C09076=1067.956,264.109,-90.042,173.798,30.770,155.599
C09077=1067.962,264.356,-90.071,173.801,30.774,155.599
C09078=1067.968,264.604,-90.100,173.804,30.779,155.600
C09079=1067.974,264.852,-90.129,173.805,30.782,155.601
C09080=1067.980,265.101,-90.157,173.808,30.786,155.601
C09081=1067.986,265.349,-90.187,173.811,30.791,155.602
C09082=1067.992,265.598,-90.216,173.813,30.794,155.603
C09083=1067.998,265.846,-90.245,173.816,30.798,155.604
C09084=1068.005,266.094,-90.274,173.819,30.803,155.604
C09085=1068.010,266.342,-90.304,173.821,30.806,155.605
C09086=1068.016,266.591,-90.332,173.823,30.811,155.606
C09087=1068.022,266.838,-90.361,173.826,30.815,155.606
C09088=1068.028,267.087,-90.390,173.829,30.818,155.607
C09089=1068.033,267.335,-90.419,173.831,30.823,155.608
C09090=1068.040,267.583,-90.449,173.834,30.827,155.609
C09091=1068.046,267.831,-90.478,173.837,30.831,155.609
C09092=1068.052,268.079,-90.507,173.838,30.835,155.610
C09093=1068.058,268.328,-90.536,173.841,30.839,155.611
C09094=1068.064,268.576,-90.565,173.844,30.842,155.611
C09095=1068.070,268.824,-90.594,173.847,30.846,155.612
C09096=1068.076,269.072,-90.623,173.849,30.851,155.613
C09097=1068.082,269.321,-90.653,173.852,30.854,155.613
C09098=1068.088,269.569,-90.682,173.855,30.859,155.614
C09099=1068.094,269.817,-90.712,173.857,30.863,155.615
C09100=1068.100,270.065,-90.741,173.860,30.867,155.616
C09101=1068.106,270.314,-90.770,173.862,30.871,155.616
C09102=1068.112,270.562,-90.799,173.864,30.875,155.617
C09103=1068.118,270.810,-90.829,173.867,30.878,155.618
C09104=1068.124,271.058,-90.859,173.870,30.883,155.618
C09105=1068.130,271.306,-90.888,173.873,30.887,155.619
C09106=1068.136,271.554,-90.917,173.875,30.891,155.620
C09107=1068.142,271.803,-90.946,173.878,30.895,155.621
C09108=1068.148,272.051,-90.976,173.881,30.899,155.621
C09109=1068.154,272.299,-91.006,173.883,30.903,155.622
C09110=1068.161,272.547,-91.035,173.886,30.907,155.623
C09111=1068.166,272.796,-91.065,173.888,30.911,155.623
C09112=1068.173,273.044,-91.094,173.891,30.915,155.624
C09113=1068.178,273.292,-91.124,173.893,30.919,155.625
C09114=1068.185,273.540,-91.153,173.896,30.923,155.626
C09115=1068.190,273.788,-91.183,173.899,30.927,155.626
C09116=1068.197,274.036,-91.213,173.901,30.931,155.627
C09117=1068.202,274.284,-91.242,173.904,30.935,155.628
C09118=1068.208,274.532,-91.271,173.907,30.939,155.628
C09119=1068.214,274.780,-91.302,173.910,30.943,155.629
C09120=1068.220,275.028,-91.331,173.912,30.947,155.630
C09121=1068.227,275.278,-91.361,173.915,30.951,155.631
C09122=1068.232,275.525,-91.391,173.918,30.955,155.631
C09123=1068.239,275.774,-91.420,173.920,30.960,155.632
C09124=1068.244,275.987,-91.446,173.922,30.963,155.633
C09125=1068.249,276.202,-91.471,173.925,30.967,155.633
C09126=1068.255,276.416,-91.497,173.927,30.970,155.634
C09127=1068.259,276.630,-91.524,173.929,30.974,155.634
C09128=1068.264,276.845,-91.549,173.931,30.977,155.635
C09129=1068.270,277.059,-91.575,173.934,30.980,155.636
C09130=1068.275,277.273,-91.600,173.936,30.984,155.636
C09131=1068.280,277.487,-91.626,173.938,30.987,155.637
C09132=1068.286,277.735,-91.657,173.941,30.992,155.638
C09133=1068.292,277.983,-91.686,173.944,30.996,155.638
C09134=1068.298,278.231,-91.716,173.947,31.000,155.639
C09135=1068.304,278.480,-91.746,173.949,31.004,155.640
C09136=1068.311,278.727,-91.776,173.952,31.008,155.640
C09137=1068.316,278.976,-91.805,173.955,31.012,155.641
C09138=1068.322,279.224,-91.836,173.957,31.016,155.642
C09139=1068.328,279.472,-91.866,173.960,31.020,155.643
C09140=1068.335,279.720,-91.896,173.963,31.024,155.643
C09141=1068.340,279.968,-91.926,173.966,31.028,155.644
C09142=1068.346,280.216,-91.956,173.968,31.032,155.645
C09143=1068.353,280.464,-91.985,173.971,31.036,155.646
C09144=1068.358,280.712,-92.016,173.974,31.040,155.646
C09145=1068.365,280.961,-92.046,173.977,31.045,155.647
C09146=1068.371,281.208,-92.077,173.978,31.048,155.648
C09147=1068.376,281.457,-92.106,173.981,31.053,155.648
C09148=1068.382,281.705,-92.137,173.984,31.056,155.649
C09149=1068.388,281.953,-92.167,173.986,31.061,155.650
C09150=1068.394,282.201,-92.198,173.989,31.065,155.651
C09151=1068.400,282.449,-92.228,173.992,31.069,155.651
C09152=1068.406,282.697,-92.257,173.995,31.073,155.652
C09153=1068.412,282.945,-92.288,173.997,31.077,155.653
C09154=1068.418,283.193,-92.318,174.000,31.081,155.654
C09155=1068.424,283.441,-92.349,174.003,31.085,155.654
C09156=1068.430,283.689,-92.379,174.006,31.090,155.655
C09157=1068.436,283.937,-92.410,174.008,31.093,155.656
C09158=1068.442,284.185,-92.440,174.011,31.098,155.656
C09159=1068.448,284.433,-92.470,174.015,31.102,155.657
C09160=1068.455,284.682,-92.501,174.017,31.106,155.658
C09161=1068.460,284.929,-92.531,174.020,31.110,155.659
C09162=1068.466,285.177,-92.562,174.023,31.114,155.659
C09163=1068.473,285.426,-92.592,174.026,31.119,155.660
C09164=1068.478,285.674,-92.623,174.028,31.122,155.661
C09165=1068.484,285.921,-92.653,174.031,31.127,155.662
C09166=1068.491,286.170,-92.684,174.034,31.131,155.662
C09167=1068.496,286.418,-92.714,174.037,31.135,155.663
C09168=1068.502,286.666,-92.745,174.039,31.139,155.664
C09169=1068.509,286.914,-92.775,174.042,31.143,155.664
C09170=1068.515,287.162,-92.805,174.045,31.147,155.665
C09171=1068.521,287.409,-92.835,174.048,31.151,155.666
C09172=1068.527,287.658,-92.866,174.050,31.155,155.667
C09173=1068.533,287.906,-92.896,174.053,31.159,155.667
C09174=1068.540,288.154,-92.928,174.056,31.164,155.668
C09175=1068.546,288.401,-92.958,174.059,31.168,155.669
C09176=1068.552,288.650,-92.989,174.061,31.172,155.670
C09177=1068.558,288.898,-93.019,174.064,31.176,155.670
C09178=1068.563,289.146,-93.050,174.067,31.180,155.671
C09179=1068.570,289.394,-93.082,174.069,31.184,155.672
C09180=1068.575,289.613,-93.108,174.072,31.188,155.673
C09181=1068.580,289.832,-93.136,174.075,31.192,155.673
C09182=1068.586,290.052,-93.163,174.078,31.195,155.674
C09183=1068.591,290.271,-93.191,174.080,31.199,155.675
C09184=1068.597,290.490,-93.217,174.082,31.203,155.675
C09185=1068.602,290.710,-93.245,174.085,31.206,155.676
C09186=1068.607,290.929,-93.272,174.088,31.210,155.676
C09187=1068.613,291.149,-93.300,174.090,31.214,155.677
C09188=1068.619,291.397,-93.330,174.092,31.218,155.678
C09189=1068.625,291.645,-93.361,174.095,31.222,155.679
C09190=1068.631,291.893,-93.393,174.099,31.226,155.679
C09191=1068.636,292.141,-93.423,174.102,31.230,155.680
C09192=1068.643,292.389,-93.454,174.104,31.235,155.681
C09193=1068.649,292.636,-93.485,174.107,31.239,155.682
C09194=1068.655,292.885,-93.517,174.110,31.243,155.682
C09195=1068.661,293.132,-93.547,174.113,31.247,155.683
C09196=1068.667,293.381,-93.578,174.115,31.252,155.684
C09197=1068.673,293.628,-93.609,174.118,31.255,155.685
C09198=1068.679,293.877,-93.640,174.121,31.260,155.685
C09199=1068.685,294.124,-93.671,174.124,31.264,155.686
C09200=1068.692,294.372,-93.703,174.127,31.268,155.687
C09201=1068.697,294.620,-93.734,174.130,31.272,155.688
C09202=1068.704,294.868,-93.765,174.133,31.277,155.688
C09203=1068.710,295.117,-93.796,174.136,31.281,155.689
C09204=1068.715,295.364,-93.827,174.138,31.285,155.690
C09205=1068.722,295.612,-93.859,174.141,31.289,155.691
C09206=1068.728,295.860,-93.889,174.144,31.293,155.692
C09207=1068.734,296.108,-93.921,174.147,31.298,155.692
C09208=1068.740,296.355,-93.952,174.150,31.302,155.693
C09209=1068.746,296.604,-93.984,174.153,31.306,155.694
C09210=1068.753,296.852,-94.015,174.156,31.310,155.695
C09211=1068.759,297.099,-94.046,174.159,31.315,155.695
C09212=1068.764,297.348,-94.077,174.161,31.319,155.696
C09213=1068.770,297.595,-94.108,174.164,31.323,155.697
C09214=1068.776,297.843,-94.140,174.167,31.327,155.698
C09215=1068.782,298.091,-94.172,174.171,31.332,155.698
C09216=1068.789,298.339,-94.204,174.173,31.336,155.699
C09217=1068.794,298.586,-94.235,174.176,31.341,155.700
C09218=1068.800,298.835,-94.267,174.179,31.345,155.701
C09219=1068.806,299.083,-94.298,174.182,31.349,155.702
C09220=1068.812,299.331,-94.330,174.184,31.354,155.702
C09221=1068.818,299.579,-94.362,174.188,31.357,155.703
C09222=1068.824,299.826,-94.393,174.191,31.362,155.704
C09223=1068.830,300.074,-94.425,174.194,31.366,155.705
C09224=1068.836,300.322,-94.457,174.196,31.370,155.705
C09225=1068.842,300.570,-94.488,174.199,31.375,155.706
C09226=1068.848,300.818,-94.520,174.202,31.379,155.707
C09227=1068.853,301.065,-94.552,174.206,31.383,155.708
C09228=1068.859,301.314,-94.584,174.208,31.388,155.709
C09229=1068.866,301.562,-94.615,174.211,31.392,155.709
C09230=1068.871,301.809,-94.647,174.214,31.396,155.710
C09231=1068.877,302.057,-94.679,174.217,31.401,155.711
C09232=1068.884,302.305,-94.710,174.220,31.405,155.712
C09233=1068.890,302.553,-94.742,174.223,31.409,155.713
C09234=1068.896,302.801,-94.774,174.226,31.414,155.713
C09235=1068.902,303.049,-94.806,174.229,31.418,155.714
C09236=1068.908,303.275,-94.835,174.232,31.422,155.715
C09237=1068.913,303.502,-94.864,174.234,31.426,155.716
C09238=1068.918,303.729,-94.893,174.237,31.430,155.716
C09239=1068.924,303.956,-94.922,174.240,31.434,155.717
C09240=1068.930,304.182,-94.952,174.243,31.438,155.718
C09241=1068.935,304.409,-94.981,174.245,31.442,155.719
C09242=1068.940,304.636,-95.010,174.248,31.446,155.719
C09243=1068.946,304.863,-95.040,174.251,31.450,155.720
C09244=1068.952,305.110,-95.071,174.254,31.455,155.721
C09245=1068.958,305.359,-95.103,174.257,31.459,155.722
C09246=1068.964,305.607,-95.135,174.259,31.463,155.722
C09247=1068.971,305.854,-95.168,174.263,31.468,155.723
C09248=1068.976,306.102,-95.200,174.266,31.472,155.724
C09249=1068.983,306.350,-95.231,174.269,31.476,155.725
C09250=1068.989,306.597,-95.264,174.271,31.480,155.726
C09251=1068.995,306.846,-95.296,174.275,31.485,155.726
C09252=1069.001,307.094,-95.328,174.278,31.489,155.727
C09253=1069.007,307.341,-95.361,174.281,31.494,155.728
C09254=1069.014,307.589,-95.392,174.284,31.498,155.729
C09255=1069.020,307.836,-95.424,174.287,31.502,155.730
C09256=1069.026,308.085,-95.456,174.290,31.507,155.730
C09257=1069.032,308.332,-95.489,174.293,31.511,155.731
C09258=1069.038,308.580,-95.521,174.297,31.516,155.732
C09259=1069.045,308.828,-95.553,174.299,31.520,155.733
C09260=1069.051,309.076,-95.585,174.302,31.524,155.734
C09261=1069.057,309.324,-95.617,174.305,31.529,155.734
C09262=1069.063,309.572,-95.650,174.309,31.533,155.735
C09263=1069.069,309.819,-95.682,174.312,31.537,155.736
C09264=1069.075,310.067,-95.715,174.314,31.542,155.737
C09265=1069.081,310.314,-95.747,174.318,31.546,155.738
C09266=1069.088,310.562,-95.779,174.321,31.550,155.738
C09267=1069.094,310.810,-95.811,174.324,31.555,155.739
C09268=1069.100,311.058,-95.843,174.326,31.559,155.740
C09269=1069.107,311.306,-95.876,174.330,31.564,155.741
C09270=1069.113,311.553,-95.909,174.333,31.568,155.742
C09271=1069.119,311.801,-95.941,174.336,31.572,155.742
C09272=1069.125,312.049,-95.974,174.340,31.577,155.743
C09273=1069.132,312.297,-96.006,174.342,31.581,155.744
C09274=1069.138,312.544,-96.038,174.345,31.585,155.745
C09275=1069.145,312.792,-96.071,174.349,31.590,155.746
C09276=1069.151,313.040,-96.104,174.352,31.595,155.747
C09277=1069.158,313.288,-96.137,174.355,31.599,155.747
C09278=1069.164,313.536,-96.169,174.358,31.603,155.748
C09279=1069.170,313.784,-96.201,174.361,31.608,155.749
C09280=1069.176,314.031,-96.234,174.364,31.612,155.750
C09281=1069.183,314.279,-96.267,174.368,31.617,155.751
C09282=1069.189,314.527,-96.300,174.370,31.621,155.751
C09283=1069.194,314.775,-96.332,174.373,31.626,155.752
C09284=1069.200,315.023,-96.365,174.377,31.630,155.753
C09285=1069.207,315.270,-96.398,174.380,31.635,155.754
C09286=1069.212,315.518,-96.431,174.383,31.640,155.755
C09287=1069.219,315.766,-96.464,174.386,31.644,155.756
C09288=1069.224,316.014,-96.497,174.389,31.649,155.757
C09289=1069.230,316.261,-96.530,174.392,31.654,155.758
C09290=1069.237,316.509,-96.563,174.396,31.658,155.758
C09291=1069.242,316.757,-96.596,174.399,31.663,155.759
C09292=1069.248,316.985,-96.626,174.401,31.666,155.760
C09293=1069.253,317.214,-96.656,174.404,31.671,155.761
C09294=1069.260,317.443,-96.687,174.407,31.675,155.762
C09295=1069.265,317.671,-96.718,174.410,31.679,155.762
C09296=1069.270,317.899,-96.749,174.413,31.684,155.763
C09297=1069.276,318.128,-96.779,174.415,31.688,155.764
C09298=1069.282,318.357,-96.810,174.418,31.692,155.765
C09299=1069.287,318.585,-96.840,174.422,31.696,155.765
C09300=1069.293,318.833,-96.873,174.425,31.701,155.766
C09301=1069.300,319.080,-96.907,174.428,31.706,155.767
C09302=1069.305,319.328,-96.940,174.431,31.710,155.768
C09303=1069.311,319.576,-96.973,174.434,31.715,155.769
C09304=1069.318,319.823,-97.005,174.437,31.720,155.770
C09305=1069.324,320.072,-97.039,174.441,31.724,155.771
C09306=1069.331,320.319,-97.073,174.444,31.729,155.772
C09307=1069.336,320.567,-97.106,174.447,31.734,155.772
C09308=1069.342,320.814,-97.139,174.450,31.738,155.773
C09309=1069.348,321.062,-97.173,174.453,31.743,155.774
C09310=1069.355,321.310,-97.206,174.457,31.748,155.775
C09311=1069.361,321.558,-97.239,174.460,31.752,155.776
C09312=1069.367,321.805,-97.273,174.463,31.757,155.777
C09313=1069.373,322.053,-97.306,174.466,31.762,155.778
C09314=1069.380,322.301,-97.339,174.469,31.766,155.779
C09315=1069.386,322.548,-97.373,174.473,31.771,155.779
C09316=1069.392,322.796,-97.406,174.476,31.776,155.780
C09317=1069.397,323.044,-97.439,174.479,31.780,155.781
C09318=1069.405,323.291,-97.473,174.482,31.785,155.782
C09319=1069.410,323.539,-97.506,174.486,31.790,155.783
C09320=1069.417,323.786,-97.540,174.489,31.794,155.784
C09321=1069.423,324.035,-97.573,174.492,31.799,155.785
C09322=1069.430,324.282,-97.607,174.495,31.804,155.786
C09323=1069.435,324.530,-97.640,174.498,31.808,155.786
C09324=1069.442,324.778,-97.674,174.502,31.813,155.787
C09325=1069.448,325.025,-97.707,174.505,31.818,155.788
C09326=1069.454,325.273,-97.741,174.509,31.823,155.789
C09327=1069.461,325.520,-97.775,174.512,31.827,155.790
C09328=1069.466,325.768,-97.809,174.515,31.832,155.791
C09329=1069.473,326.015,-97.842,174.518,31.837,155.792
C09330=1069.480,326.263,-97.877,174.521,31.841,155.793
C09331=1069.486,326.511,-97.909,174.525,31.846,155.794
C09332=1069.492,326.759,-97.944,174.528,31.850,155.795
C09333=1069.499,327.006,-97.977,174.531,31.855,155.795
C09334=1069.505,327.254,-98.011,174.534,31.860,155.796
C09335=1069.511,327.502,-98.045,174.538,31.865,155.797
C09336=1069.518,327.749,-98.078,174.541,31.869,155.798
C09337=1069.524,327.997,-98.112,174.545,31.874,155.799
C09338=1069.530,328.244,-98.146,174.547,31.879,155.800
C09339=1069.537,328.492,-98.180,174.551,31.884,155.801
C09340=1069.543,328.739,-98.214,174.554,31.888,155.802
C09341=1069.550,328.987,-98.248,174.558,31.893,155.803
C09342=1069.555,329.235,-98.281,174.561,31.898,155.804
C09343=1069.562,329.483,-98.316,174.565,31.903,155.804
C09344=1069.568,329.730,-98.349,174.567,31.908,155.805
C09345=1069.575,329.978,-98.383,174.571,31.912,155.806
C09346=1069.582,330.226,-98.417,174.574,31.917,155.807
C09347=1069.588,330.473,-98.451,174.578,31.922,155.808
C09348=1069.594,330.698,-98.482,174.581,31.926,155.809
C09349=1069.600,330.924,-98.514,174.584,31.931,155.810
C09350=1069.605,331.150,-98.544,174.587,31.935,155.811
C09351=1069.611,331.376,-98.576,174.590,31.940,155.811
C09352=1069.617,331.601,-98.606,174.593,31.944,155.812
C09353=1069.622,331.826,-98.638,174.596,31.948,155.813
C09354=1069.629,332.052,-98.669,174.600,31.953,155.814
C09355=1069.634,332.277,-98.700,174.603,31.957,155.815
C09356=1069.640,332.525,-98.734,174.605,31.962,155.816
C09357=1069.646,332.773,-98.769,174.609,31.967,155.817
C09358=1069.652,333.019,-98.804,174.612,31.972,155.818
C09359=1069.659,333.267,-98.838,174.616,31.977,155.819
C09360=1069.665,333.515,-98.872,174.619,31.982,155.820
C09361=1069.671,333.763,-98.906,174.623,31.987,155.820
C09362=1069.677,334.011,-98.941,174.626,31.992,155.822
C09363=1069.684,334.257,-98.976,174.629,31.997,155.822
C09364=1069.690,334.505,-99.010,174.633,32.002,155.823
C09365=1069.697,334.753,-99.044,174.636,32.007,155.824
C09366=1069.702,335.000,-99.079,174.640,32.012,155.825
C09367=1069.709,335.248,-99.114,174.643,32.017,155.826
C09368=1069.715,335.495,-99.148,174.646,32.022,155.827
C09369=1069.721,335.743,-99.182,174.650,32.027,155.828
C09370=1069.728,335.990,-99.217,174.653,32.032,155.829
C09371=1069.734,336.238,-99.251,174.657,32.037,155.830
C09372=1069.741,336.486,-99.286,174.660,32.041,155.831
C09373=1069.747,336.733,-99.321,174.664,32.047,155.832
C09374=1069.753,336.980,-99.355,174.667,32.052,155.833
C09375=1069.760,337.228,-99.390,174.670,32.056,155.834
C09376=1069.766,337.476,-99.425,174.674,32.062,155.835
C09377=1069.773,337.723,-99.460,174.677,32.067,155.836
C09378=1069.778,337.971,-99.494,174.681,32.072,155.837
C09379=1069.785,338.218,-99.529,174.685,32.077,155.838
C09380=1069.792,338.466,-99.564,174.688,32.082,155.839
C09381=1069.798,338.713,-99.599,174.691,32.087,155.840
C09382=1069.803,338.961,-99.634,174.695,32.093,155.841
C09383=1069.810,339.208,-99.669,174.698,32.097,155.842
C09384=1069.816,339.455,-99.704,174.702,32.103,155.843
C09385=1069.823,339.703,-99.738,174.705,32.107,155.844
C09386=1069.829,339.951,-99.774,174.709,32.113,155.845
C09387=1069.836,340.198,-99.809,174.713,32.118,155.846
C09388=1069.842,340.445,-99.843,174.715,32.123,155.847
C09389=1069.848,340.693,-99.879,174.719,32.128,155.848
C09390=1069.854,340.940,-99.914,174.723,32.133,155.849
C09391=1069.861,341.188,-99.948,174.726,32.138,155.850
C09392=1069.868,341.436,-99.983,174.730,32.143,155.851
C09393=1069.873,341.683,-100.019,174.734,32.149,155.852
C09394=1069.880,341.930,-100.054,174.737,32.154,155.853
C09395=1069.886,342.177,-100.089,174.740,32.159,155.854
C09396=1069.892,342.426,-100.124,174.744,32.164,155.855
C09397=1069.899,342.673,-100.159,174.747,32.170,155.856
C09398=1069.906,342.920,-100.194,174.751,32.175,155.857
C09399=1069.911,343.167,-100.230,174.755,32.180,155.858
C09400=1069.918,343.415,-100.265,174.758,32.185,155.859
C09401=1069.925,343.662,-100.300,174.762,32.190,155.860
C09402=1069.931,343.910,-100.336,174.765,32.195,155.861
C09403=1069.938,344.157,-100.371,174.769,32.201,155.862
C09404=1069.946,344.493,-100.418,174.774,32.208,155.863
C09405=1069.954,344.828,-100.467,174.779,32.215,155.865
C09406=1069.963,345.164,-100.515,174.784,32.223,155.866
C09407=1069.972,345.500,-100.563,174.789,32.230,155.868
C09408=1069.978,345.748,-100.598,174.791,32.235,155.869
C09409=1069.985,345.995,-100.634,174.795,32.240,155.870
C09410=1069.991,346.243,-100.670,174.799,32.246,155.871
C09411=1069.998,346.490,-100.705,174.803,32.251,155.872
C09412=1070.004,346.738,-100.741,174.806,32.256,155.873
C09413=1070.010,346.984,-100.776,174.810,32.262,155.874
C09414=1070.016,347.231,-100.812,174.814,32.267,155.875
C09415=1070.022,347.479,-100.848,174.818,32.273,155.876
C09416=1070.029,347.726,-100.883,174.820,32.278,155.877
C09417=1070.035,347.974,-100.919,174.824,32.283,155.878
C09418=1070.042,348.221,-100.955,174.828,32.289,155.879
C09419=1070.048,348.468,-100.990,174.832,32.294,155.880
C09420=1070.054,348.716,-101.026,174.835,32.299,155.881
C09421=1070.061,348.963,-101.062,174.839,32.305,155.883
C09422=1070.067,349.211,-101.098,174.843,32.310,155.884
C09423=1070.073,349.458,-101.133,174.847,32.316,155.885
C09424=1070.081,349.706,-101.169,174.849,32.321,155.886
C09425=1070.087,349.953,-101.205,174.853,32.326,155.887
C09426=1070.093,350.200,-101.242,174.857,32.332,155.888
C09427=1070.100,350.448,-101.277,174.861,32.338,155.889
C09428=1070.106,350.695,-101.313,174.865,32.343,155.890
C09429=1070.112,350.942,-101.349,174.868,32.348,155.891
C09430=1070.119,351.190,-101.385,174.872,32.354,155.892
C09431=1070.126,351.437,-101.421,174.876,32.360,155.893
C09432=1070.135,351.794,-101.473,174.882,32.367,155.895
C09433=1070.145,352.152,-101.525,174.886,32.376,155.897
C09434=1070.154,352.509,-101.578,174.892,32.384,155.898
C09435=1070.163,352.867,-101.630,174.897,32.391,155.900
C09436=1070.169,353.114,-101.665,174.901,32.397,155.901
C09437=1070.176,353.361,-101.702,174.905,32.403,155.902
C09438=1070.182,353.609,-101.738,174.909,32.409,155.903
C09439=1070.189,353.856,-101.775,174.912,32.414,155.904
C09440=1070.195,354.103,-101.812,174.916,32.420,155.906
C09441=1070.201,354.351,-101.847,174.919,32.426,155.907
C09442=1070.208,354.598,-101.884,174.923,32.431,155.908
C09443=1070.214,354.845,-101.920,174.927,32.437,155.909
C09444=1070.220,355.092,-101.957,174.931,32.443,155.910
C09445=1070.227,355.340,-101.993,174.935,32.448,155.911
C09446=1070.234,355.587,-102.030,174.938,32.454,155.912
C09447=1070.240,355.834,-102.066,174.942,32.460,155.914
C09448=1070.246,356.081,-102.103,174.946,32.465,155.915
C09449=1070.253,356.329,-102.140,174.950,32.471,155.916
C09450=1070.260,356.576,-102.175,174.954,32.477,155.917
C09451=1070.267,356.823,-102.212,174.958,32.482,155.918
C09452=1070.273,357.070,-102.248,174.962,32.488,155.919
C09453=1070.280,357.317,-102.285,174.965,32.494,155.920
C09454=1070.286,357.565,-102.322,174.969,32.500,155.922
C09455=1070.293,357.812,-102.358,174.972,32.505,155.923
C09456=1070.298,358.037,-102.391,174.976,32.511,155.924
C09457=1070.305,358.262,-102.425,174.980,32.516,155.925
C09458=1070.310,358.487,-102.459,174.983,32.521,155.926
C09459=1070.316,358.712,-102.492,174.987,32.527,155.927
C09460=1070.322,358.937,-102.526,174.990,32.532,155.928
C09461=1070.328,359.161,-102.558,174.994,32.537,155.929
C09462=1070.334,359.386,-102.592,174.997,32.542,155.930
C09463=1070.340,359.611,-102.625,175.001,32.548,155.931
C09464=1070.346,359.858,-102.662,175.005,32.554,155.932
C09465=1070.353,360.106,-102.699,175.009,32.559,155.934
C09466=1070.359,360.352,-102.736,175.013,32.565,155.935
C09467=1070.366,360.600,-102.773,175.016,32.571,155.936
C09468=1070.373,360.847,-102.810,175.020,32.577,155.937
C09469=1070.379,361.093,-102.847,175.024,32.583,155.938
C09470=1070.386,361.341,-102.884,175.028,32.589,155.940
C09471=1070.392,361.588,-102.921,175.031,32.595,155.941
C09472=1070.399,361.836,-102.958,175.035,32.601,155.942
C09473=1070.406,362.082,-102.995,175.039,32.607,155.943
C09474=1070.412,362.329,-103.032,175.043,32.612,155.945
C09475=1070.419,362.576,-103.069,175.047,32.619,155.946
C09476=1070.425,362.824,-103.106,175.051,32.625,155.947
C09477=1070.432,363.071,-103.144,175.055,32.630,155.948
C09478=1070.438,363.318,-103.180,175.059,32.637,155.950
C09479=1070.445,363.565,-103.219,175.063,32.643,155.951
C09480=1070.451,363.812,-103.255,175.067,32.649,155.952
C09481=1070.458,364.060,-103.292,175.071,32.655,155.953
C09482=1070.465,364.306,-103.330,175.075,32.661,155.954
C09483=1070.471,364.554,-103.367,175.079,32.667,155.956
C09484=1070.478,364.800,-103.404,175.083,32.673,155.957
C09485=1070.484,365.048,-103.442,175.086,32.679,155.958
C09486=1070.491,365.294,-103.479,175.090,32.685,155.959
C09487=1070.497,365.542,-103.517,175.094,32.691,155.961
C09488=1070.504,365.789,-103.554,175.098,32.698,155.962
C09489=1070.511,366.036,-103.592,175.102,32.704,155.963
C09490=1070.517,366.283,-103.629,175.106,32.710,155.965
C09491=1070.524,366.530,-103.667,175.110,32.716,155.966
C09492=1070.530,366.777,-103.705,175.115,32.722,155.967
C09493=1070.537,367.024,-103.743,175.119,32.729,155.968
C09494=1070.543,367.271,-103.779,175.123,32.735,155.970
C09495=1070.550,367.519,-103.817,175.127,32.741,155.971
C09496=1070.557,367.766,-103.855,175.131,32.747,155.972
C09497=1070.563,368.012,-103.893,175.135,32.754,155.974
C09498=1070.570,368.260,-103.930,175.139,32.760,155.975
C09499=1070.576,368.506,-103.968,175.143,32.766,155.976
C09500=1070.583,368.753,-104.006,175.147,32.773,155.977
C09501=1070.590,369.000,-104.044,175.151,32.779,155.979
C09502=1070.597,369.247,-104.081,175.155,32.785,155.980
C09503=1070.603,369.494,-104.120,175.159,32.792,155.981
C09504=1070.610,369.742,-104.158,175.163,32.798,155.983
C09505=1070.616,369.988,-104.195,175.167,32.804,155.984
C09506=1070.623,370.235,-104.233,175.172,32.811,155.985
C09507=1070.630,370.482,-104.271,175.176,32.817,155.987
C09508=1070.637,370.729,-104.309,175.180,32.823,155.988
C09509=1070.643,370.976,-104.346,175.184,32.830,155.989
C09510=1070.650,371.223,-104.385,175.188,32.836,155.991
C09511=1070.657,371.470,-104.423,175.192,32.842,155.992
C09512=1070.663,371.703,-104.459,175.196,32.849,155.993
C09513=1070.670,371.937,-104.494,175.200,32.854,155.995
C09514=1070.675,372.170,-104.531,175.204,32.861,155.996
C09515=1070.682,372.403,-104.567,175.208,32.867,155.997
C09516=1070.689,372.636,-104.602,175.212,32.873,155.998
C09517=1070.695,372.870,-104.638,175.216,32.879,156.000
C09518=1070.702,373.104,-104.675,175.220,32.885,156.001
C09519=1070.708,373.337,-104.711,175.223,32.891,156.002
C09520=1070.714,373.583,-104.750,175.228,32.898,156.004
C09521=1070.720,373.831,-104.788,175.232,32.904,156.005
C09522=1070.728,374.077,-104.826,175.236,32.911,156.006
C09523=1070.735,374.325,-104.864,175.240,32.918,156.008
C09524=1070.741,374.572,-104.903,175.244,32.924,156.009
C09525=1070.748,374.818,-104.941,175.248,32.931,156.011
C09526=1070.754,375.065,-104.980,175.253,32.938,156.012
C09527=1070.761,375.312,-105.018,175.257,32.945,156.013
C09528=1070.768,375.559,-105.057,175.261,32.951,156.015
C09529=1070.774,375.806,-105.095,175.265,32.958,156.016
C09530=1070.781,376.053,-105.134,175.269,32.965,156.018
C09531=1070.788,376.300,-105.173,175.274,32.971,156.019
C09532=1070.794,376.546,-105.212,175.278,32.978,156.020
C09533=1070.802,376.792,-105.250,175.282,32.985,156.022
C09534=1070.808,377.040,-105.288,175.286,32.991,156.023
C09535=1070.815,377.287,-105.327,175.290,32.998,156.025
C09536=1070.822,377.534,-105.366,175.295,33.005,156.026
C09537=1070.829,377.780,-105.404,175.299,33.012,156.028
C09538=1070.835,378.027,-105.443,175.304,33.019,156.029
C09539=1070.842,378.274,-105.482,175.308,33.025,156.030
C09540=1070.849,378.521,-105.521,175.313,33.032,156.032
C09541=1070.856,378.768,-105.560,175.317,33.039,156.033
C09542=1070.863,379.015,-105.599,175.321,33.046,156.035
C09543=1070.869,379.261,-105.637,175.325,33.053,156.036
C09544=1070.876,379.508,-105.676,175.330,33.060,156.038
C09545=1070.883,379.755,-105.715,175.334,33.067,156.039
C09546=1070.890,380.002,-105.754,175.338,33.074,156.041
C09547=1070.897,380.249,-105.793,175.343,33.080,156.042
C09548=1070.904,380.495,-105.832,175.347,33.087,156.044
C09549=1070.911,380.742,-105.871,175.351,33.094,156.045
C09550=1070.917,380.989,-105.910,175.355,33.101,156.047
C09551=1070.925,381.236,-105.949,175.360,33.108,156.048
C09552=1070.932,381.483,-105.988,175.364,33.115,156.050
C09553=1070.938,381.729,-106.028,175.368,33.122,156.051
C09554=1070.945,381.976,-106.067,175.374,33.129,156.053
C09555=1070.952,382.223,-106.106,175.378,33.137,156.054
C09556=1070.959,382.469,-106.145,175.382,33.143,156.056
C09557=1070.965,382.716,-106.185,175.387,33.151,156.057
C09558=1070.972,382.963,-106.224,175.391,33.158,156.059
C09559=1070.979,383.209,-106.263,175.395,33.165,156.060
C09560=1070.985,383.456,-106.303,175.400,33.172,156.062
C09561=1070.992,383.703,-106.342,175.404,33.180,156.063
C09562=1071.000,383.950,-106.382,175.408,33.186,156.065
C09563=1071.006,384.197,-106.422,175.413,33.194,156.067
C09564=1071.013,384.443,-106.461,175.417,33.201,156.068
C09565=1071.020,384.690,-106.500,175.422,33.208,156.070
C09566=1071.026,384.936,-106.540,175.427,33.216,156.071
C09567=1071.034,385.183,-106.580,175.431,33.223,156.073
C09568=1071.041,385.432,-106.619,175.436,33.231,156.074
C09569=1071.048,385.683,-106.660,175.440,33.238,156.076
C09570=1071.054,385.932,-106.699,175.444,33.245,156.078
C09571=1071.062,386.181,-106.740,175.449,33.253,156.079
C09572=1071.068,386.428,-106.779,175.453,33.260,156.081
C09573=1071.075,386.675,-106.819,175.458,33.267,156.082
C09574=1071.083,386.922,-106.859,175.463,33.275,156.084
C09575=1071.090,387.168,-106.899,175.468,33.282,156.086
C09576=1071.096,387.414,-106.939,175.472,33.290,156.087
C09577=1071.103,387.661,-106.979,175.477,33.297,156.089
C09578=1071.110,387.908,-107.019,175.481,33.304,156.090
C09579=1071.117,388.155,-107.058,175.485,33.312,156.092
C09580=1071.125,388.402,-107.098,175.490,33.320,156.094
C09581=1071.131,388.648,-107.138,175.495,33.327,156.095
C09582=1071.138,388.894,-107.178,175.500,33.334,156.097
C09583=1071.145,389.141,-107.218,175.504,33.342,156.099
C09584=1071.153,389.387,-107.258,175.509,33.349,156.100
C09585=1071.160,389.634,-107.299,175.513,33.357,156.102
C09586=1071.167,389.880,-107.338,175.518,33.365,156.104
C09587=1071.173,390.127,-107.379,175.523,33.372,156.105
C09588=1071.181,390.374,-107.419,175.528,33.380,156.107
C09589=1071.188,390.620,-107.458,175.532,33.388,156.109
C09590=1071.195,390.867,-107.499,175.537,33.395,156.110
C09591=1071.202,391.113,-107.539,175.541,33.403,156.112
C09592=1071.209,391.360,-107.579,175.546,33.411,156.114
C09593=1071.216,391.607,-107.620,175.551,33.418,156.115
C09594=1071.223,391.853,-107.661,175.556,33.426,156.117
C09595=1071.230,392.099,-107.700,175.560,33.434,156.119
C09596=1071.237,392.347,-107.741,175.565,33.442,156.121
C09597=1071.244,392.592,-107.782,175.570,33.450,156.122
C09598=1071.251,392.839,-107.822,175.574,33.458,156.124
C09599=1071.258,393.085,-107.862,175.580,33.465,156.126
C09600=1071.265,393.333,-107.903,175.584,33.473,156.127
C09601=1071.273,393.579,-107.944,175.589,33.481,156.129
C09602=1071.280,393.825,-107.984,175.593,33.489,156.131
C09603=1071.287,394.072,-108.025,175.598,33.497,156.133
C09604=1071.293,394.318,-108.065,175.603,33.504,156.134
C09605=1071.300,394.565,-108.106,175.608,33.513,156.136
C09606=1071.308,394.812,-108.148,175.613,33.521,156.138
C09607=1071.315,395.058,-108.187,175.617,33.529,156.140
C09608=1071.322,395.304,-108.228,175.623,33.537,156.141
C09609=1071.329,395.551,-108.270,175.627,33.545,156.143
C09610=1071.336,395.797,-108.310,175.632,33.553,156.145
C09611=1071.343,396.044,-108.351,175.637,33.561,156.147
C09612=1071.350,396.291,-108.392,175.642,33.569,156.149
C09613=1071.357,396.537,-108.433,175.647,33.577,156.150
C09614=1071.364,396.783,-108.474,175.652,33.586,156.152
C09615=1071.372,397.030,-108.516,175.656,33.594,156.154
C09616=1071.380,397.276,-108.556,175.662,33.602,156.156
C09617=1071.386,397.523,-108.596,175.666,33.610,156.158
C09618=1071.393,397.769,-108.638,175.671,33.619,156.160
C09619=1071.401,398.016,-108.679,175.676,33.627,156.161
C09620=1071.408,398.262,-108.720,175.681,33.635,156.163
C09621=1071.415,398.509,-108.761,175.686,33.643,156.165
C09622=1071.422,398.755,-108.802,175.691,33.652,156.167
C09623=1071.429,399.001,-108.845,175.696,33.660,156.169
C09624=1071.437,399.267,-108.888,175.702,33.669,156.171
C09625=1071.444,399.532,-108.933,175.707,33.678,156.173
C09626=1071.452,399.797,-108.978,175.712,33.687,156.175
C09627=1071.460,400.062,-109.023,175.718,33.696,156.177
C09628=1071.467,400.309,-109.064,175.722,33.705,156.179
C09629=1071.474,400.555,-109.105,175.727,33.713,156.181
C09630=1071.482,400.801,-109.147,175.733,33.722,156.183
C09631=1071.489,401.048,-109.188,175.738,33.730,156.185
C09632=1071.496,401.295,-109.229,175.742,33.739,156.187
C09633=1071.503,401.541,-109.272,175.747,33.747,156.189
C09634=1071.511,401.787,-109.313,175.753,33.756,156.190
C09635=1071.518,402.034,-109.354,175.758,33.765,156.192
C09636=1071.525,402.280,-109.396,175.763,33.773,156.194
C09637=1071.533,402.527,-109.438,175.768,33.782,156.196
C09638=1071.540,402.773,-109.480,175.773,33.790,156.198
C09639=1071.547,403.019,-109.521,175.778,33.799,156.200
C09640=1071.555,403.265,-109.563,175.784,33.808,156.202
C09641=1071.562,403.512,-109.605,175.789,33.817,156.204
C09642=1071.569,403.758,-109.647,175.794,33.826,156.206
C09643=1071.576,404.004,-109.689,175.799,33.834,156.208
C09644=1071.584,404.251,-109.730,175.804,33.843,156.210
C09645=1071.591,404.498,-109.773,175.810,33.852,156.212
C09646=1071.599,404.744,-109.815,175.815,33.861,156.214
C09647=1071.606,404.990,-109.857,175.820,33.870,156.216
C09648=1071.613,405.237,-109.899,175.825,33.879,156.218
C09649=1071.620,405.483,-109.941,175.830,33.888,156.220
C09650=1071.627,405.729,-109.983,175.835,33.897,156.222
C09651=1071.635,405.975,-110.025,175.841,33.906,156.224
C09652=1071.642,406.222,-110.068,175.846,33.915,156.226
C09653=1071.650,406.468,-110.110,175.852,33.924,156.229
C09654=1071.657,406.714,-110.153,175.857,33.933,156.231
C09655=1071.664,406.960,-110.195,175.862,33.942,156.233
C09656=1071.672,407.207,-110.238,175.868,33.951,156.235
C09657=1071.679,407.453,-110.279,175.873,33.961,156.237
C09658=1071.686,407.699,-110.322,175.879,33.970,156.239
C09659=1071.693,407.946,-110.365,175.884,33.979,156.241
C09660=1071.701,408.192,-110.407,175.889,33.989,156.243
C09661=1071.708,408.438,-110.450,175.894,33.998,156.245
C09662=1071.715,408.684,-110.493,175.900,34.007,156.248
C09663=1071.723,408.930,-110.535,175.905,34.016,156.250
C09664=1071.730,409.177,-110.578,175.910,34.026,156.252
C09665=1071.737,409.423,-110.621,175.916,34.035,156.254
C09666=1071.746,409.670,-110.663,175.921,34.044,156.256
C09667=1071.753,409.916,-110.706,175.927,34.054,156.258
C09668=1071.760,410.162,-110.749,175.933,34.063,156.260
C09669=1071.768,410.408,-110.791,175.939,34.073,156.263
C09670=1071.775,410.654,-110.834,175.944,34.082,156.265
C09671=1071.782,410.901,-110.877,175.950,34.092,156.267
C09672=1071.790,411.146,-110.920,175.955,34.101,156.269
C09673=1071.798,411.393,-110.963,175.961,34.111,156.271
C09674=1071.805,411.639,-111.006,175.966,34.121,156.274
C09675=1071.813,411.886,-111.048,175.972,34.130,156.276
C09676=1071.820,412.131,-111.092,175.977,34.140,156.278
C09677=1071.828,412.378,-111.135,175.983,34.149,156.280
C09678=1071.835,412.624,-111.178,175.988,34.159,156.283
C09679=1071.843,412.870,-111.221,175.995,34.169,156.285
C09680=1071.851,413.138,-111.268,176.000,34.179,156.287
C09681=1071.860,413.408,-111.315,176.007,34.190,156.290
C09682=1071.868,413.677,-111.363,176.013,34.201,156.292
C09683=1071.877,413.945,-111.410,176.019,34.212,156.295
C09684=1071.885,414.191,-111.453,176.025,34.221,156.297
C09685=1071.892,414.437,-111.497,176.031,34.231,156.299
C09686=1071.899,414.684,-111.539,176.037,34.241,156.302
C09687=1071.907,414.930,-111.583,176.042,34.251,156.304
C09688=1071.915,415.176,-111.627,176.048,34.261,156.306
C09689=1071.922,415.421,-111.671,176.054,34.271,156.309
C09690=1071.930,415.668,-111.714,176.060,34.282,156.311
C09691=1071.938,415.914,-111.758,176.066,34.291,156.313
C09692=1071.945,416.160,-111.801,176.071,34.302,156.316
C09693=1071.953,416.406,-111.845,176.077,34.312,156.318
C09694=1071.961,416.652,-111.889,176.084,34.322,156.321
C09695=1071.968,416.898,-111.933,176.089,34.332,156.323
C09696=1071.976,417.144,-111.976,176.095,34.343,156.325
C09697=1071.983,417.390,-112.020,176.102,34.353,156.328
C09698=1071.991,417.636,-112.064,176.107,34.363,156.330
C09699=1071.999,417.882,-112.108,176.113,34.373,156.333
C09700=1072.007,418.128,-112.152,176.120,34.384,156.335
C09701=1072.014,418.374,-112.196,176.125,34.394,156.338
C09702=1072.022,418.620,-112.240,176.131,34.405,156.340
C09703=1072.030,418.866,-112.284,176.138,34.415,156.343
C09704=1072.038,419.112,-112.328,176.143,34.426,156.345
C09705=1072.045,419.358,-112.372,176.150,34.436,156.347
C09706=1072.053,419.604,-112.416,176.156,34.447,156.350
C09707=1072.061,419.850,-112.460,176.161,34.457,156.352
C09708=1072.069,420.096,-112.504,176.168,34.468,156.355
C09709=1072.077,420.342,-112.549,176.174,34.478,156.357
C09710=1072.085,420.588,-112.593,176.181,34.489,156.360
C09711=1072.093,420.834,-112.638,176.186,34.500,156.363
C09712=1072.101,421.079,-112.682,176.193,34.510,156.365
C09713=1072.109,421.326,-112.726,176.199,34.521,156.368
C09714=1072.116,421.572,-112.771,176.206,34.532,156.370
C09715=1072.124,421.818,-112.815,176.211,34.543,156.373
C09716=1072.131,422.064,-112.860,176.218,34.554,156.375
C09717=1072.139,422.309,-112.904,176.224,34.564,156.378
C09718=1072.148,422.555,-112.949,176.231,34.576,156.381
C09719=1072.155,422.801,-112.994,176.236,34.586,156.383
C09720=1072.163,423.046,-113.038,176.243,34.598,156.386
C09721=1072.170,423.292,-113.083,176.249,34.609,156.389
C09722=1072.179,423.538,-113.128,176.256,34.620,156.391
C09723=1072.186,423.784,-113.173,176.262,34.631,156.394
C09724=1072.194,424.029,-113.218,176.269,34.642,156.396
C09725=1072.203,424.276,-113.262,176.275,34.653,156.399
C09726=1072.210,424.522,-113.307,176.281,34.664,156.402
C09727=1072.219,424.767,-113.352,176.288,34.676,156.405
C09728=1072.226,425.013,-113.397,176.295,34.687,156.407
C09729=1072.234,425.258,-113.442,176.301,34.698,156.410
C09730=1072.242,425.505,-113.488,176.308,34.710,156.413
C09731=1072.251,425.750,-113.533,176.315,34.721,156.415
C09732=1072.258,425.996,-113.578,176.321,34.733,156.418
C09733=1072.267,426.242,-113.623,176.327,34.744,156.421
C09734=1072.275,426.487,-113.669,176.334,34.755,156.424
C09735=1072.283,426.733,-113.713,176.340,34.767,156.426
C09736=1072.292,427.021,-113.767,176.348,34.780,156.430
C09737=1072.301,427.308,-113.819,176.357,34.794,156.433
C09738=1072.311,427.595,-113.873,176.365,34.807,156.436
C09739=1072.321,427.882,-113.926,176.372,34.821,156.440
C09740=1072.329,428.128,-113.972,176.379,34.833,156.443
C09741=1072.337,428.374,-114.017,176.386,34.845,156.445
C09742=1072.344,428.620,-114.062,176.393,34.856,156.448
C09743=1072.353,428.865,-114.108,176.400,34.868,156.451
C09744=1072.361,429.110,-114.154,176.406,34.880,156.454
C09745=1072.369,429.356,-114.200,176.413,34.892,156.457
C09746=1072.377,429.602,-114.246,176.420,34.904,156.460
C09747=1072.385,429.847,-114.291,176.427,34.916,156.463
C09748=1072.394,430.093,-114.337,176.434,34.928,156.466
C09749=1072.401,430.339,-114.383,176.441,34.940,156.469
C09750=1072.410,430.584,-114.429,176.448,34.952,156.472
C09751=1072.418,430.830,-114.475,176.455,34.964,156.475
C09752=1072.427,431.075,-114.520,176.462,34.976,156.477
C09753=1072.435,431.321,-114.567,176.468,34.988,156.480
C09754=1072.443,431.566,-114.613,176.475,35.001,156.484
C09755=1072.451,431.812,-114.660,176.483,35.013,156.487
C09756=1072.460,432.058,-114.706,176.490,35.025,156.490
C09757=1072.467,432.303,-114.752,176.497,35.038,156.493
C09758=1072.476,432.549,-114.798,176.504,35.051,156.496
C09759=1072.484,432.795,-114.845,176.511,35.063,156.499
C09760=1072.492,433.039,-114.891,176.518,35.075,156.502
C09761=1072.501,433.285,-114.938,176.526,35.088,156.505
C09762=1072.509,433.531,-114.984,176.533,35.100,156.508
C09763=1072.517,433.776,-115.030,176.541,35.113,156.511
C09764=1072.525,434.021,-115.077,176.548,35.126,156.514
C09765=1072.534,434.267,-115.124,176.555,35.138,156.517
C09766=1072.543,434.512,-115.170,176.563,35.151,156.521
C09767=1072.550,434.757,-115.217,176.570,35.164,156.524
C09768=1072.558,435.003,-115.264,176.577,35.177,156.527
C09769=1072.567,435.249,-115.311,176.584,35.190,156.530
C09770=1072.575,435.494,-115.357,176.592,35.203,156.533
C09771=1072.584,435.740,-115.404,176.600,35.215,156.537
C09772=1072.592,435.985,-115.451,176.607,35.228,156.540
C09773=1072.601,436.230,-115.498,176.615,35.241,156.543
C09774=1072.610,436.475,-115.545,176.622,35.255,156.546
C09775=1072.618,436.721,-115.592,176.629,35.268,156.550
C09776=1072.627,436.966,-115.640,176.638,35.281,156.553
C09777=1072.635,437.212,-115.687,176.645,35.294,156.556
C09778=1072.644,437.457,-115.733,176.652,35.307,156.559
C09779=1072.652,437.702,-115.781,176.660,35.320,156.563
C09780=1072.661,437.948,-115.827,176.668,35.334,156.566
C09781=1072.670,438.192,-115.875,176.676,35.347,156.569
C09782=1072.678,438.438,-115.922,176.683,35.360,156.573
C09783=1072.687,438.683,-115.970,176.692,35.374,156.576
C09784=1072.695,438.928,-116.017,176.699,35.388,156.580
C09785=1072.704,439.173,-116.065,176.706,35.401,156.583
C09786=1072.712,439.419,-116.112,176.715,35.415,156.586
C09787=1072.721,439.664,-116.159,176.722,35.428,156.590
C09788=1072.730,439.910,-116.208,176.731,35.442,156.593
C09789=1072.738,440.155,-116.255,176.738,35.456,156.597
C09790=1072.747,440.399,-116.303,176.747,35.470,156.600
C09791=1072.755,440.645,-116.351,176.755,35.483,156.604
C09792=1072.768,440.976,-116.415,176.766,35.502,156.608
C09793=1072.779,441.309,-116.480,176.777,35.521,156.613
C09794=1072.791,441.640,-116.545,176.787,35.540,156.618
C09795=1072.803,441.973,-116.611,176.798,35.559,156.623
C09796=1072.812,442.217,-116.659,176.807,35.573,156.627
C09797=1072.820,442.462,-116.707,176.815,35.587,156.630
C09798=1072.829,442.708,-116.755,176.823,35.602,156.634
C09799=1072.838,442.952,-116.803,176.832,35.616,156.637
C09800=1072.847,443.197,-116.851,176.840,35.630,156.641
C09801=1072.856,443.443,-116.900,176.848,35.645,156.645
C09802=1072.865,443.688,-116.947,176.856,35.659,156.649
C09803=1072.874,443.933,-116.996,176.865,35.673,156.652
C09804=1072.882,444.177,-117.045,176.874,35.688,156.656
C09805=1072.891,444.423,-117.093,176.881,35.702,156.660
C09806=1072.900,444.668,-117.142,176.890,35.717,156.663
C09807=1072.909,444.913,-117.191,176.899,35.732,156.667
C09808=1072.918,445.157,-117.239,176.908,35.747,156.671
C09809=1072.927,445.402,-117.288,176.916,35.762,156.675
C09810=1072.936,445.648,-117.337,176.925,35.776,156.679
C09811=1072.945,445.892,-117.386,176.933,35.791,156.683
C09812=1072.954,446.137,-117.435,176.942,35.806,156.686
C09813=1072.963,446.382,-117.483,176.951,35.821,156.690
C09814=1072.972,446.627,-117.532,176.960,35.836,156.694
C09815=1072.981,446.872,-117.582,176.968,35.851,156.698
C09816=1072.990,447.118,-117.631,176.977,35.866,156.702
C09817=1072.999,447.361,-117.680,176.986,35.882,156.706
C09818=1073.008,447.607,-117.729,176.995,35.896,156.710
C09819=1073.017,447.852,-117.778,177.003,35.912,156.714
C09820=1073.027,448.096,-117.827,177.011,35.927,156.718
C09821=1073.036,448.339,-117.876,177.018,35.942,156.722
C09822=1073.046,448.584,-117.925,177.026,35.957,156.725
C09823=1073.056,448.828,-117.973,177.033,35.972,156.729
C09824=1073.068,449.074,-118.021,177.040,35.985,156.733
C09825=1073.081,449.318,-118.068,177.047,35.999,156.737
C09826=1073.096,449.563,-118.113,177.054,36.012,156.740
C09827=1073.111,449.809,-118.158,177.059,36.025,156.743
C09828=1072.758,449.807,-118.403,177.043,36.171,156.782
C09829=1072.743,449.561,-118.358,177.036,36.158,156.779
C09830=1072.728,449.316,-118.313,177.031,36.145,156.775
C09831=1072.714,449.071,-118.266,177.024,36.132,156.772
C09832=1072.703,448.826,-118.218,177.016,36.118,156.768
C09833=1072.692,448.582,-118.169,177.009,36.104,156.764
C09834=1072.683,448.337,-118.121,177.002,36.089,156.761
C09835=1072.673,448.093,-118.072,176.993,36.074,156.757
C09836=1072.663,447.849,-118.023,176.985,36.059,156.753
C09837=1072.654,447.606,-117.974,176.977,36.043,156.749
C09838=1072.645,447.360,-117.924,176.968,36.028,156.745
C09839=1072.636,447.116,-117.875,176.959,36.013,156.741
C09840=1072.627,446.870,-117.826,176.950,35.998,156.737
C09841=1072.617,446.625,-117.777,176.941,35.983,156.733
C09842=1072.609,446.381,-117.728,176.932,35.968,156.729
C09843=1072.599,446.136,-117.678,176.924,35.953,156.725
C09844=1072.590,445.891,-117.629,176.915,35.938,156.721
C09845=1072.581,445.647,-117.581,176.906,35.923,156.717
C09846=1072.572,445.401,-117.532,176.897,35.908,156.714
C09847=1072.563,445.156,-117.483,176.888,35.894,156.710
C09848=1072.555,444.911,-117.434,176.880,35.879,156.706
C09849=1072.545,444.666,-117.386,176.871,35.864,156.702
C09850=1072.537,444.421,-117.338,176.862,35.849,156.698
C09851=1072.528,444.176,-117.288,176.854,35.835,156.695
C09852=1072.518,443.931,-117.240,176.846,35.821,156.691
C09853=1072.510,443.686,-117.191,176.837,35.806,156.687
C09854=1072.501,443.440,-117.143,176.828,35.792,156.684
C09855=1072.492,443.196,-117.095,176.820,35.777,156.680
C09856=1072.483,442.952,-117.046,176.811,35.763,156.676
C09857=1072.474,442.706,-116.998,176.803,35.748,156.672
C09858=1072.466,442.461,-116.950,176.795,35.735,156.669
C09859=1072.456,442.216,-116.901,176.786,35.721,156.665
C09860=1072.448,441.971,-116.853,176.778,35.706,156.662
C09861=1072.436,441.657,-116.792,176.767,35.688,156.657
C09862=1072.426,441.344,-116.730,176.757,35.670,156.652
C09863=1072.414,441.029,-116.669,176.747,35.652,156.648
C09864=1072.403,440.716,-116.607,176.736,35.635,156.643
C09865=1072.394,440.472,-116.560,176.728,35.621,156.640
C09866=1072.385,440.226,-116.511,176.719,35.607,156.636
C09867=1072.376,439.981,-116.464,176.712,35.593,156.633
C09868=1072.368,439.736,-116.416,176.704,35.580,156.629
C09869=1072.359,439.491,-116.369,176.696,35.566,156.626
C09870=1072.351,439.246,-116.321,176.688,35.553,156.623
C09871=1072.343,439.000,-116.274,176.679,35.539,156.619
C09872=1072.333,438.754,-116.226,176.672,35.525,156.616
C09873=1072.324,438.509,-116.178,176.664,35.512,156.612
C09874=1072.316,438.264,-116.130,176.656,35.499,156.609
C09875=1072.308,438.019,-116.084,176.648,35.485,156.605
C09876=1072.299,437.774,-116.036,176.641,35.472,156.602
C09877=1072.290,437.528,-115.990,176.632,35.458,156.599
C09878=1072.281,437.283,-115.942,176.625,35.445,156.595
C09879=1072.272,437.037,-115.895,176.618,35.432,156.592
C09880=1072.264,436.792,-115.847,176.610,35.419,156.589
C09881=1072.256,436.547,-115.800,176.602,35.406,156.586
C09882=1072.247,436.301,-115.754,176.594,35.393,156.582
C09883=1072.238,436.056,-115.706,176.587,35.380,156.579
C09884=1072.230,435.811,-115.660,176.579,35.367,156.576
C09885=1072.222,435.566,-115.613,176.571,35.354,156.573
C09886=1072.213,435.320,-115.566,176.564,35.341,156.569
C09887=1072.205,435.075,-115.520,176.556,35.328,156.566
C09888=1072.197,434.830,-115.471,176.549,35.315,156.563
C09889=1072.188,434.584,-115.425,176.542,35.303,156.560
C09890=1072.180,434.339,-115.378,176.534,35.290,156.557
C09891=1072.171,434.093,-115.331,176.527,35.277,156.553
C09892=1072.163,433.848,-115.285,176.520,35.265,156.550
C09893=1072.155,433.602,-115.239,176.511,35.252,156.547
C09894=1072.146,433.357,-115.192,176.504,35.239,156.544
C09895=1072.138,433.111,-115.145,176.497,35.227,156.541
C09896=1072.130,432.866,-115.099,176.490,35.215,156.538
C09897=1072.121,432.621,-115.052,176.482,35.202,156.535
C09898=1072.113,432.375,-115.006,176.475,35.189,156.532
C09899=1072.105,432.130,-114.960,176.468,35.177,156.529
C09900=1072.097,431.884,-114.913,176.461,35.165,156.526
C09901=1072.088,431.638,-114.867,176.454,35.153,156.523
C09902=1072.080,431.393,-114.821,176.446,35.140,156.519
C09903=1072.072,431.147,-114.775,176.439,35.128,156.516
C09904=1072.064,430.902,-114.728,176.433,35.116,156.514
C09905=1072.056,430.656,-114.683,176.426,35.104,156.511
C09906=1072.047,430.410,-114.637,176.419,35.091,156.508
C09907=1072.038,430.165,-114.590,176.412,35.079,156.505
C09908=1072.031,429.919,-114.545,176.404,35.068,156.502
C09909=1072.023,429.673,-114.499,176.397,35.056,156.499
C09910=1072.014,429.428,-114.454,176.390,35.043,156.496
C09911=1072.006,429.183,-114.407,176.383,35.032,156.493
C09912=1071.998,428.937,-114.361,176.376,35.020,156.490
C09913=1071.990,428.691,-114.315,176.370,35.008,156.487
C09914=1071.981,428.446,-114.270,176.363,34.996,156.484
C09915=1071.974,428.201,-114.225,176.356,34.984,156.481
C09916=1071.965,427.954,-114.179,176.349,34.972,156.478
C09917=1071.956,427.666,-114.125,176.341,34.959,156.475
C09918=1071.946,427.377,-114.071,176.333,34.945,156.472
C09919=1071.937,427.088,-114.018,176.325,34.932,156.469
C09920=1071.927,426.798,-113.965,176.317,34.918,156.465
C09921=1071.919,426.553,-113.920,176.310,34.907,156.462
C09922=1071.911,426.308,-113.874,176.304,34.895,156.460
C09923=1071.902,426.062,-113.829,176.297,34.884,156.457
C09924=1071.895,425.816,-113.784,176.290,34.872,156.454
C09925=1071.887,425.571,-113.739,176.284,34.861,156.451
C09926=1071.879,425.324,-113.694,176.277,34.850,156.449
C09927=1071.870,425.079,-113.649,176.270,34.838,156.446
C09928=1071.863,424.833,-113.604,176.264,34.827,156.443
C09929=1071.855,424.588,-113.559,176.257,34.816,156.440
C09930=1071.847,424.341,-113.513,176.250,34.805,156.438
C09931=1071.838,424.096,-113.468,176.245,34.793,156.435
C09932=1071.831,423.850,-113.423,176.238,34.782,156.432
C09933=1071.823,423.604,-113.379,176.232,34.771,156.430
C09934=1071.815,423.359,-113.334,176.225,34.760,156.427
C09935=1071.807,423.112,-113.289,176.218,34.749,156.424
C09936=1071.799,422.866,-113.244,176.212,34.738,156.422
C09937=1071.791,422.620,-113.199,176.205,34.727,156.419
C09938=1071.783,422.375,-113.155,176.199,34.716,156.416
C09939=1071.776,422.129,-113.109,176.193,34.705,156.414
C09940=1071.768,421.883,-113.065,176.187,34.694,156.411
C09941=1071.759,421.638,-113.021,176.180,34.683,156.409
C09942=1071.752,421.392,-112.976,176.174,34.673,156.406
C09943=1071.744,421.146,-112.931,176.167,34.662,156.404
C09944=1071.736,420.899,-112.888,176.161,34.651,156.401
C09945=1071.728,420.654,-112.843,176.155,34.640,156.398
C09946=1071.721,420.408,-112.798,176.149,34.630,156.396
C09947=1071.713,420.162,-112.754,176.142,34.619,156.393
C09948=1071.705,419.916,-112.710,176.136,34.608,156.391
C09949=1071.697,419.670,-112.665,176.130,34.598,156.388
C09950=1071.689,419.424,-112.622,176.124,34.587,156.386
C09951=1071.681,419.178,-112.578,176.118,34.577,156.383
C09952=1071.673,418.933,-112.533,176.111,34.566,156.381
C09953=1071.666,418.686,-112.489,176.105,34.556,156.378
C09954=1071.658,418.440,-112.445,176.100,34.545,156.376
C09955=1071.650,418.194,-112.401,176.093,34.535,156.373
C09956=1071.642,417.949,-112.357,176.087,34.525,156.371
C09957=1071.635,417.702,-112.313,176.082,34.515,156.369
C09958=1071.627,417.457,-112.269,176.075,34.504,156.366
C09959=1071.619,417.210,-112.225,176.069,34.494,156.364
C09960=1071.611,416.964,-112.182,176.063,34.484,156.361
C09961=1071.603,416.718,-112.137,176.057,34.473,156.359
C09962=1071.596,416.473,-112.094,176.051,34.463,156.356
C09963=1071.589,416.226,-112.050,176.045,34.453,156.354
C09964=1071.581,415.980,-112.006,176.040,34.443,156.352
C09965=1071.574,415.734,-111.962,176.033,34.433,156.349
C09966=1071.566,415.488,-111.919,176.027,34.423,156.347
C09967=1071.558,415.242,-111.875,176.022,34.413,156.345
C09968=1071.551,414.996,-111.832,176.016,34.403,156.342
C09969=1071.543,414.750,-111.788,176.009,34.393,156.340
C09970=1071.535,414.504,-111.745,176.004,34.383,156.338
C09971=1071.527,414.257,-111.702,175.998,34.373,156.335
C09972=1071.520,414.012,-111.658,175.993,34.363,156.333
C09973=1071.511,413.741,-111.611,175.986,34.352,156.330
C09974=1071.503,413.471,-111.563,175.979,34.341,156.328
C09975=1071.494,413.200,-111.516,175.974,34.331,156.325
C09976=1071.486,412.930,-111.468,175.967,34.320,156.323
C09977=1071.478,412.684,-111.425,175.961,34.311,156.321
C09978=1071.471,412.438,-111.382,175.956,34.301,156.318
C09979=1071.463,412.191,-111.339,175.950,34.291,156.316
C09980=1071.455,411.945,-111.295,175.945,34.281,156.314
C09981=1071.448,411.699,-111.253,175.938,34.272,156.312
C09982=1071.440,411.452,-111.209,175.932,34.262,156.309
C09983=1071.433,411.207,-111.166,175.927,34.252,156.307
C09984=1071.424,410.960,-111.124,175.921,34.243,156.305
C09985=1071.417,410.714,-111.081,175.916,34.233,156.303
C09986=1071.410,410.467,-111.038,175.910,34.224,156.301
C09987=1071.402,410.222,-110.995,175.905,34.214,156.298
C09988=1071.395,409.976,-110.952,175.899,34.205,156.296
C09989=1071.387,409.729,-110.909,175.894,34.196,156.294
C09990=1071.380,409.483,-110.866,175.888,34.186,156.292
C09991=1071.372,409.237,-110.824,175.883,34.177,156.290
C09992=1071.365,408.991,-110.781,175.877,34.167,156.288
C09993=1071.357,408.745,-110.739,175.872,34.158,156.285
C09994=1071.350,408.498,-110.696,175.866,34.149,156.283
C09995=1071.343,408.252,-110.653,175.861,34.140,156.281
C09996=1071.335,408.006,-110.611,175.855,34.130,156.279
//INST
///DATE 2021/06/17 10:55
///ATTR SC,RW,RJ
////FRAME ROBOT
///GROUP1 RB1
NOP
MOVL C00000 V=800.0 PL=0
MOVL C00001 V=800.0 PL=0
MOVL C00002 V=800.0 PL=0
MOVL C00003 V=800.0 PL=0
MOVL C00004 V=800.0 PL=0
MOVL C00005 V=800.0 PL=0
MOVL C00006 V=800.0 PL=0
MOVL C00007 V=800.0 PL=0
MOVL C00008 V=800.0 PL=0
MOVL C00009 V=800.0 PL=0
MOVL C00010 V=800.0 PL=0
MOVL C00011 V=800.0 PL=0
MOVL C00012 V=800.0 PL=0
MOVL C00013 V=800.0 PL=0
MOVL C00014 V=800.0 PL=0
MOVL C00015 V=800.0 PL=0
MOVL C00016 V=800.0 PL=0
MOVL C00017 V=800.0 PL=0
MOVL C00018 V=800.0 PL=0
MOVL C00019 V=800.0 PL=0
MOVL C00020 V=800.0 PL=0
MOVL C00021 V=800.0 PL=0
MOVL C00022 V=800.0 PL=0
MOVL C00023 V=800.0 PL=0
MOVL C00024 V=800.0 PL=0
MOVL C00025 V=800.0 PL=0
MOVL C00026 V=800.0 PL=0
MOVL C00027 V=800.0 PL=0
MOVL C00028 V=800.0 PL=0
MOVL C00029 V=800.0 PL=0
MOVL C00030 V=800.0 PL=0
MOVL C00031 V=800.0 PL=0
MOVL C00032 V=800.0 PL=0
MOVL C00033 V=800.0 PL=0
MOVL C00034 V=800.0 PL=0
MOVL C00035 V=800.0 PL=0
MOVL C00036 V=800.0 PL=0
MOVL C00037 V=800.0 PL=0
MOVL C00038 V=800.0 PL=0
MOVL C00039 V=800.0 PL=0
MOVL C00040 V=800.0 PL=0
MOVL C00041 V=800.0 PL=0
MOVL C00042 V=800.0 PL=0
MOVL C00043 V=800.0 PL=0
MOVL C00044 V=800.0 PL=0
MOVL C00045 V=800.0 PL=0
MOVL C00046 V=800.0 PL=0
MOVL C00047 V=800.0 PL=0
MOVL C00048 V=800.0 PL=0
MOVL C00049 V=800.0 PL=0
MOVL C00050 V=800.0 PL=0
MOVL C00051 V=800.0 PL=0
MOVL C00052 V=800.0 PL=0
MOVL C00053 V=800.0 PL=0
MOVL C00054 V=800.0 PL=0
MOVL C00055 V=800.0 PL=0
MOVL C00056 V=800.0 PL=0
MOVL C00057 V=800.0 PL=0
MOVL C00058 V=800.0 PL=0
MOVL C00059 V=800.0 PL=0
MOVL C00060 V=800.0 PL=0
MOVL C00061 V=800.0 PL=0
MOVL C00062 V=800.0 PL=0
MOVL C00063 V=800.0 PL=0
MOVL C00064 V=800.0 PL=0
MOVL C00065 V=800.0 PL=0
MOVL C00066 V=800.0 PL=0
MOVL C00067 V=800.0 PL=0
MOVL C00068 V=800.0 PL=0
MOVL C00069 V=800.0 PL=0
MOVL C00070 V=800.0 PL=0
MOVL C00071 V=800.0 PL=0
MOVL C00072 V=800.0 PL=0
MOVL C00073 V=800.0 PL=0
MOVL C00074 V=800.0 PL=0
MOVL C00075 V=800.0 PL=0
MOVL C00076 V=800.0 PL=0
MOVL C00077 V=800.0 PL=0
MOVL C00078 V=800.0 PL=0
MOVL C00079 V=800.0 PL=0
MOVL C00080 V=800.0 PL=0
MOVL C00081 V=800.0 PL=0
MOVL C00082 V=800.0 PL=0
MOVL C00083 V=800.0 PL=0
MOVL C00084 V=800.0 PL=0
MOVL C00085 V=800.0 PL=0
MOVL C00086 V=800.0 PL=0
MOVL C00087 V=800.0 PL=0
MOVL C00088 V=800.0 PL=0
MOVL C00089 V=800.0 PL=0
MOVL C00090 V=800.0 PL=0
MOVL C00091 V=800.0 PL=0
MOVL C00092 V=800.0 PL=0
MOVL C00093 V=800.0 PL=0
MOVL C00094 V=800.0 PL=0
MOVL C00095 V=800.0 PL=0
MOVL C00096 V=800.0 PL=0
MOVL C00097 V=800.0 PL=0
MOVL C00098 V=800.0 PL=0
MOVL C00099 V=800.0 PL=0
MOVL C00100 V=800.0 PL=0
MOVL C00101 V=800.0 PL=0
MOVL C00102 V=800.0 PL=0
MOVL C00103 V=800.0 PL=0
MOVL C00104 V=800.0 PL=0
MOVL C00105 V=800.0 PL=0
MOVL C00106 V=800.0 PL=0
MOVL C00107 V=800.0 PL=0
MOVL C00108 V=800.0 PL=0
MOVL C00109 V=800.0 PL=0
MOVL C00110 V=800.0 PL=0
MOVL C00111 V=800.0 PL=0
MOVL C00112 V=800.0 PL=0
MOVL C00113 V=800.0 PL=0
MOVL C00114 V=800.0 PL=0
MOVL C00115 V=800.0 PL=0
MOVL C00116 V=800.0 PL=0
MOVL C00117 V=800.0 PL=0
MOVL C00118 V=800.0 PL=0
MOVL C00119 V=800.0 PL=0
MOVL C00120 V=800.0 PL=0
MOVL C00121 V=800.0 PL=0
MOVL C00122 V=800.0 PL=0
MOVL C00123 V=800.0 PL=0
MOVL C00124 V=800.0 PL=0
MOVL C00125 V=800.0 PL=0
MOVL C00126 V=800.0 PL=0
MOVL C00127 V=800.0 PL=0
MOVL C00128 V=800.0 PL=0
MOVL C00129 V=800.0 PL=0
MOVL C00130 V=800.0 PL=0
MOVL C00131 V=800.0 PL=0
MOVL C00132 V=800.0 PL=0
MOVL C00133 V=800.0 PL=0
MOVL C00134 V=800.0 PL=0
MOVL C00135 V=800.0 PL=0
MOVL C00136 V=800.0 PL=0
MOVL C00137 V=800.0 PL=0
MOVL C00138 V=800.0 PL=0
MOVL C00139 V=800.0 PL=0
MOVL C00140 V=800.0 PL=0
MOVL C00141 V=800.0 PL=0
MOVL C00142 V=800.0 PL=0
MOVL C00143 V=800.0 PL=0
MOVL C00144 V=800.0 PL=0
MOVL C00145 V=800.0 PL=0
MOVL C00146 V=800.0 PL=0
MOVL C00147 V=800.0 PL=0
MOVL C00148 V=800.0 PL=0
MOVL C00149 V=800.0 PL=0
MOVL C00150 V=800.0 PL=0
MOVL C00151 V=800.0 PL=0
MOVL C00152 V=800.0 PL=0
MOVL C00153 V=800.0 PL=0
MOVL C00154 V=800.0 PL=0
MOVL C00155 V=800.0 PL=0
MOVL C00156 V=800.0 PL=0
MOVL C00157 V=800.0 PL=0
MOVL C00158 V=800.0 PL=0
MOVL C00159 V=800.0 PL=0
MOVL C00160 V=800.0 PL=0
MOVL C00161 V=800.0 PL=0
MOVL C00162 V=800.0 PL=0
MOVL C00163 V=800.0 PL=0
MOVL C00164 V=800.0 PL=0
MOVL C00165 V=800.0 PL=0
MOVL C00166 V=800.0 PL=0
MOVL C00167 V=800.0 PL=0
MOVL C00168 V=800.0 PL=0
MOVL C00169 V=800.0 PL=0
MOVL C00170 V=800.0 PL=0
MOVL C00171 V=800.0 PL=0
MOVL C00172 V=800.0 PL=0
MOVL C00173 V=800.0 PL=0
MOVL C00174 V=800.0 PL=0
MOVL C00175 V=800.0 PL=0
MOVL C00176 V=800.0 PL=0
MOVL C00177 V=800.0 PL=0
MOVL C00178 V=800.0 PL=0
MOVL C00179 V=800.0 PL=0
MOVL C00180 V=800.0 PL=0
MOVL C00181 V=800.0 PL=0
MOVL C00182 V=800.0 PL=0
MOVL C00183 V=800.0 PL=0
MOVL C00184 V=800.0 PL=0
MOVL C00185 V=800.0 PL=0
MOVL C00186 V=800.0 PL=0
MOVL C00187 V=800.0 PL=0
MOVL C00188 V=800.0 PL=0
MOVL C00189 V=800.0 PL=0
MOVL C00190 V=800.0 PL=0
MOVL C00191 V=800.0 PL=0
MOVL C00192 V=800.0 PL=0
MOVL C00193 V=800.0 PL=0
MOVL C00194 V=800.0 PL=0
MOVL C00195 V=800.0 PL=0
MOVL C00196 V=800.0 PL=0
MOVL C00197 V=800.0 PL=0
MOVL C00198 V=800.0 PL=0
MOVL C00199 V=800.0 PL=0
MOVL C00200 V=800.0 PL=0
MOVL C00201 V=800.0 PL=0
MOVL C00202 V=800.0 PL=0
MOVL C00203 V=800.0 PL=0
MOVL C00204 V=800.0 PL=0
MOVL C00205 V=800.0 PL=0
MOVL C00206 V=800.0 PL=0
MOVL C00207 V=800.0 PL=0
MOVL C00208 V=800.0 PL=0
MOVL C00209 V=800.0 PL=0
MOVL C00210 V=800.0 PL=0
MOVL C00211 V=800.0 PL=0
MOVL C00212 V=800.0 PL=0
MOVL C00213 V=800.0 PL=0
MOVL C00214 V=800.0 PL=0
MOVL C00215 V=800.0 PL=0
MOVL C00216 V=800.0 PL=0
MOVL C00217 V=800.0 PL=0
MOVL C00218 V=800.0 PL=0
MOVL C00219 V=800.0 PL=0
MOVL C00220 V=800.0 PL=0
MOVL C00221 V=800.0 PL=0
MOVL C00222 V=800.0 PL=0
MOVL C00223 V=800.0 PL=0
MOVL C00224 V=800.0 PL=0
MOVL C00225 V=800.0 PL=0
MOVL C00226 V=800.0 PL=0
MOVL C00227 V=800.0 PL=0
MOVL C00228 V=800.0 PL=0
MOVL C00229 V=800.0 PL=0
MOVL C00230 V=800.0 PL=0
MOVL C00231 V=800.0 PL=0
MOVL C00232 V=800.0 PL=0
MOVL C00233 V=800.0 PL=0
MOVL C00234 V=800.0 PL=0
MOVL C00235 V=800.0 PL=0
MOVL C00236 V=800.0 PL=0
MOVL C00237 V=800.0 PL=0
MOVL C00238 V=800.0 PL=0
MOVL C00239 V=800.0 PL=0
MOVL C00240 V=800.0 PL=0
MOVL C00241 V=800.0 PL=0
MOVL C00242 V=800.0 PL=0
MOVL C00243 V=800.0 PL=0
MOVL C00244 V=800.0 PL=0
MOVL C00245 V=800.0 PL=0
MOVL C00246 V=800.0 PL=0
MOVL C00247 V=800.0 PL=0
MOVL C00248 V=800.0 PL=0
MOVL C00249 V=800.0 PL=0
MOVL C00250 V=800.0 PL=0
MOVL C00251 V=800.0 PL=0
MOVL C00252 V=800.0 PL=0
MOVL C00253 V=800.0 PL=0
MOVL C00254 V=800.0 PL=0
MOVL C00255 V=800.0 PL=0
MOVL C00256 V=800.0 PL=0
MOVL C00257 V=800.0 PL=0
MOVL C00258 V=800.0 PL=0
MOVL C00259 V=800.0 PL=0
MOVL C00260 V=800.0 PL=0
MOVL C00261 V=800.0 PL=0
MOVL C00262 V=800.0 PL=0
MOVL C00263 V=800.0 PL=0
MOVL C00264 V=800.0 PL=0
MOVL C00265 V=800.0 PL=0
MOVL C00266 V=800.0 PL=0
MOVL C00267 V=800.0 PL=0
MOVL C00268 V=800.0 PL=0
MOVL C00269 V=800.0 PL=0
MOVL C00270 V=800.0 PL=0
MOVL C00271 V=800.0 PL=0
MOVL C00272 V=800.0 PL=0
MOVL C00273 V=800.0 PL=0
MOVL C00274 V=800.0 PL=0
MOVL C00275 V=800.0 PL=0
MOVL C00276 V=800.0 PL=0
MOVL C00277 V=800.0 PL=0
MOVL C00278 V=800.0 PL=0
MOVL C00279 V=800.0 PL=0
MOVL C00280 V=800.0 PL=0
MOVL C00281 V=800.0 PL=0
MOVL C00282 V=800.0 PL=0
MOVL C00283 V=800.0 PL=0
MOVL C00284 V=800.0 PL=0
MOVL C00285 V=800.0 PL=0
MOVL C00286 V=800.0 PL=0
MOVL C00287 V=800.0 PL=0
MOVL C00288 V=800.0 PL=0
MOVL C00289 V=800.0 PL=0
MOVL C00290 V=800.0 PL=0
MOVL C00291 V=800.0 PL=0
MOVL C00292 V=800.0 PL=0
MOVL C00293 V=800.0 PL=0
MOVL C00294 V=800.0 PL=0
MOVL C00295 V=800.0 PL=0
MOVL C00296 V=800.0 PL=0
MOVL C00297 V=800.0 PL=0
MOVL C00298 V=800.0 PL=0
MOVL C00299 V=800.0 PL=0
MOVL C00300 V=800.0 PL=0
MOVL C00301 V=800.0 PL=0
MOVL C00302 V=800.0 PL=0
MOVL C00303 V=800.0 PL=0
MOVL C00304 V=800.0 PL=0
MOVL C00305 V=800.0 PL=0
MOVL C00306 V=800.0 PL=0
MOVL C00307 V=800.0 PL=0
MOVL C00308 V=800.0 PL=0
MOVL C00309 V=800.0 PL=0
MOVL C00310 V=800.0 PL=0
MOVL C00311 V=800.0 PL=0
MOVL C00312 V=800.0 PL=0
MOVL C00313 V=800.0 PL=0
MOVL C00314 V=800.0 PL=0
MOVL C00315 V=800.0 PL=0
MOVL C00316 V=800.0 PL=0
MOVL C00317 V=800.0 PL=0
MOVL C00318 V=800.0 PL=0
MOVL C00319 V=800.0 PL=0
MOVL C00320 V=800.0 PL=0
MOVL C00321 V=800.0 PL=0
MOVL C00322 V=800.0 PL=0
MOVL C00323 V=800.0 PL=0
MOVL C00324 V=800.0 PL=0
MOVL C00325 V=800.0 PL=0
MOVL C00326 V=800.0 PL=0
MOVL C00327 V=800.0 PL=0
MOVL C00328 V=800.0 PL=0
MOVL C00329 V=800.0 PL=0
MOVL C00330 V=800.0 PL=0
MOVL C00331 V=800.0 PL=0
MOVL C00332 V=800.0 PL=0
MOVL C00333 V=800.0 PL=0
MOVL C00334 V=800.0 PL=0
MOVL C00335 V=800.0 PL=0
MOVL C00336 V=800.0 PL=0
MOVL C00337 V=800.0 PL=0
MOVL C00338 V=800.0 PL=0
MOVL C00339 V=800.0 PL=0
MOVL C00340 V=800.0 PL=0
MOVL C00341 V=800.0 PL=0
MOVL C00342 V=800.0 PL=0
MOVL C00343 V=800.0 PL=0
MOVL C00344 V=800.0 PL=0
MOVL C00345 V=800.0 PL=0
MOVL C00346 V=800.0 PL=0
MOVL C00347 V=800.0 PL=0
MOVL C00348 V=800.0 PL=0
MOVL C00349 V=800.0 PL=0
MOVL C00350 V=800.0 PL=0
MOVL C00351 V=800.0 PL=0
MOVL C00352 V=800.0 PL=0
MOVL C00353 V=800.0 PL=0
MOVL C00354 V=800.0 PL=0
MOVL C00355 V=800.0 PL=0
MOVL C00356 V=800.0 PL=0
MOVL C00357 V=800.0 PL=0
MOVL C00358 V=800.0 PL=0
MOVL C00359 V=800.0 PL=0
MOVL C00360 V=800.0 PL=0
MOVL C00361 V=800.0 PL=0
MOVL C00362 V=800.0 PL=0
MOVL C00363 V=800.0 PL=0
MOVL C00364 V=800.0 PL=0
MOVL C00365 V=800.0 PL=0
MOVL C00366 V=800.0 PL=0
MOVL C00367 V=800.0 PL=0
MOVL C00368 V=800.0 PL=0
MOVL C00369 V=800.0 PL=0
MOVL C00370 V=800.0 PL=0
MOVL C00371 V=800.0 PL=0
MOVL C00372 V=800.0 PL=0
MOVL C00373 V=800.0 PL=0
MOVL C00374 V=800.0 PL=0
MOVL C00375 V=800.0 PL=0
MOVL C00376 V=800.0 PL=0
MOVL C00377 V=800.0 PL=0
MOVL C00378 V=800.0 PL=0
MOVL C00379 V=800.0 PL=0
MOVL C00380 V=800.0 PL=0
MOVL C00381 V=800.0 PL=0
MOVL C00382 V=800.0 PL=0
MOVL C00383 V=800.0 PL=0
MOVL C00384 V=800.0 PL=0
MOVL C00385 V=800.0 PL=0
MOVL C00386 V=800.0 PL=0
MOVL C00387 V=800.0 PL=0
MOVL C00388 V=800.0 PL=0
MOVL C00389 V=800.0 PL=0
MOVL C00390 V=800.0 PL=0
MOVL C00391 V=800.0 PL=0
MOVL C00392 V=800.0 PL=0
MOVL C00393 V=800.0 PL=0
MOVL C00394 V=800.0 PL=0
MOVL C00395 V=800.0 PL=0
MOVL C00396 V=800.0 PL=0
MOVL C00397 V=800.0 PL=0
MOVL C00398 V=800.0 PL=0
MOVL C00399 V=800.0 PL=0
MOVL C00400 V=800.0 PL=0
MOVL C00401 V=800.0 PL=0
MOVL C00402 V=800.0 PL=0
MOVL C00403 V=800.0 PL=0
MOVL C00404 V=800.0 PL=0
MOVL C00405 V=800.0 PL=0
MOVL C00406 V=800.0 PL=0
MOVL C00407 V=800.0 PL=0
MOVL C00408 V=800.0 PL=0
MOVL C00409 V=800.0 PL=0
MOVL C00410 V=800.0 PL=0
MOVL C00411 V=800.0 PL=0
MOVL C00412 V=800.0 PL=0
MOVL C00413 V=800.0 PL=0
MOVL C00414 V=800.0 PL=0
MOVL C00415 V=800.0 PL=0
MOVL C00416 V=800.0 PL=0
MOVL C00417 V=800.0 PL=0
MOVL C00418 V=800.0 PL=0
MOVL C00419 V=800.0 PL=0
MOVL C00420 V=800.0 PL=0
MOVL C00421 V=800.0 PL=0
MOVL C00422 V=800.0 PL=0
MOVL C00423 V=800.0 PL=0
MOVL C00424 V=800.0 PL=0
MOVL C00425 V=800.0 PL=0
MOVL C00426 V=800.0 PL=0
MOVL C00427 V=800.0 PL=0
MOVL C00428 V=800.0 PL=0
MOVL C00429 V=800.0 PL=0
MOVL C00430 V=800.0 PL=0
MOVL C00431 V=800.0 PL=0
MOVL C00432 V=800.0 PL=0
MOVL C00433 V=800.0 PL=0
MOVL C00434 V=800.0 PL=0
MOVL C00435 V=800.0 PL=0
MOVL C00436 V=800.0 PL=0
MOVL C00437 V=800.0 PL=0
MOVL C00438 V=800.0 PL=0
MOVL C00439 V=800.0 PL=0
MOVL C00440 V=800.0 PL=0
MOVL C00441 V=800.0 PL=0
MOVL C00442 V=800.0 PL=0
MOVL C00443 V=800.0 PL=0
MOVL C00444 V=800.0 PL=0
MOVL C00445 V=800.0 PL=0
MOVL C00446 V=800.0 PL=0
MOVL C00447 V=800.0 PL=0
MOVL C00448 V=800.0 PL=0
MOVL C00449 V=800.0 PL=0
MOVL C00450 V=800.0 PL=0
MOVL C00451 V=800.0 PL=0
MOVL C00452 V=800.0 PL=0
MOVL C00453 V=800.0 PL=0
MOVL C00454 V=800.0 PL=0
MOVL C00455 V=800.0 PL=0
MOVL C00456 V=800.0 PL=0
MOVL C00457 V=800.0 PL=0
MOVL C00458 V=800.0 PL=0
MOVL C00459 V=800.0 PL=0
MOVL C00460 V=800.0 PL=0
MOVL C00461 V=800.0 PL=0
MOVL C00462 V=800.0 PL=0
MOVL C00463 V=800.0 PL=0
MOVL C00464 V=800.0 PL=0
MOVL C00465 V=800.0 PL=0
MOVL C00466 V=800.0 PL=0
MOVL C00467 V=800.0 PL=0
MOVL C00468 V=800.0 PL=0
MOVL C00469 V=800.0 PL=0
MOVL C00470 V=800.0 PL=0
MOVL C00471 V=800.0 PL=0
MOVL C00472 V=800.0 PL=0
MOVL C00473 V=800.0 PL=0
MOVL C00474 V=800.0 PL=0
MOVL C00475 V=800.0 PL=0
MOVL C00476 V=800.0 PL=0
MOVL C00477 V=800.0 PL=0
MOVL C00478 V=800.0 PL=0
MOVL C00479 V=800.0 PL=0
MOVL C00480 V=800.0 PL=0
MOVL C00481 V=800.0 PL=0
MOVL C00482 V=800.0 PL=0
MOVL C00483 V=800.0 PL=0
MOVL C00484 V=800.0 PL=0
MOVL C00485 V=800.0 PL=0
MOVL C00486 V=800.0 PL=0
MOVL C00487 V=800.0 PL=0
MOVL C00488 V=800.0 PL=0
MOVL C00489 V=800.0 PL=0
MOVL C00490 V=800.0 PL=0
MOVL C00491 V=800.0 PL=0
MOVL C00492 V=800.0 PL=0
MOVL C00493 V=800.0 PL=0
MOVL C00494 V=800.0 PL=0
MOVL C00495 V=800.0 PL=0
MOVL C00496 V=800.0 PL=0
MOVL C00497 V=800.0 PL=0
MOVL C00498 V=800.0 PL=0
MOVL C00499 V=800.0 PL=0
MOVL C00500 V=800.0 PL=0
MOVL C00501 V=800.0 PL=0
MOVL C00502 V=800.0 PL=0
MOVL C00503 V=800.0 PL=0
MOVL C00504 V=800.0 PL=0
MOVL C00505 V=800.0 PL=0
MOVL C00506 V=800.0 PL=0
MOVL C00507 V=800.0 PL=0
MOVL C00508 V=800.0 PL=0
MOVL C00509 V=800.0 PL=0
MOVL C00510 V=800.0 PL=0
MOVL C00511 V=800.0 PL=0
MOVL C00512 V=800.0 PL=0
MOVL C00513 V=800.0 PL=0
MOVL C00514 V=800.0 PL=0
MOVL C00515 V=800.0 PL=0
MOVL C00516 V=800.0 PL=0
MOVL C00517 V=800.0 PL=0
MOVL C00518 V=800.0 PL=0
MOVL C00519 V=800.0 PL=0
MOVL C00520 V=800.0 PL=0
MOVL C00521 V=800.0 PL=0
MOVL C00522 V=800.0 PL=0
MOVL C00523 V=800.0 PL=0
MOVL C00524 V=800.0 PL=0
MOVL C00525 V=800.0 PL=0
MOVL C00526 V=800.0 PL=0
MOVL C00527 V=800.0 PL=0
MOVL C00528 V=800.0 PL=0
MOVL C00529 V=800.0 PL=0
MOVL C00530 V=800.0 PL=0
MOVL C00531 V=800.0 PL=0
MOVL C00532 V=800.0 PL=0
MOVL C00533 V=800.0 PL=0
MOVL C00534 V=800.0 PL=0
MOVL C00535 V=800.0 PL=0
MOVL C00536 V=800.0 PL=0
MOVL C00537 V=800.0 PL=0
MOVL C00538 V=800.0 PL=0
MOVL C00539 V=800.0 PL=0
MOVL C00540 V=800.0 PL=0
MOVL C00541 V=800.0 PL=0
MOVL C00542 V=800.0 PL=0
MOVL C00543 V=800.0 PL=0
MOVL C00544 V=800.0 PL=0
MOVL C00545 V=800.0 PL=0
MOVL C00546 V=800.0 PL=0
MOVL C00547 V=800.0 PL=0
MOVL C00548 V=800.0 PL=0
MOVL C00549 V=800.0 PL=0
MOVL C00550 V=800.0 PL=0
MOVL C00551 V=800.0 PL=0
MOVL C00552 V=800.0 PL=0
MOVL C00553 V=800.0 PL=0
MOVL C00554 V=800.0 PL=0
MOVL C00555 V=800.0 PL=0
MOVL C00556 V=800.0 PL=0
MOVL C00557 V=800.0 PL=0
MOVL C00558 V=800.0 PL=0
MOVL C00559 V=800.0 PL=0
MOVL C00560 V=800.0 PL=0
MOVL C00561 V=800.0 PL=0
MOVL C00562 V=800.0 PL=0
MOVL C00563 V=800.0 PL=0
MOVL C00564 V=800.0 PL=0
MOVL C00565 V=800.0 PL=0
MOVL C00566 V=800.0 PL=0
MOVL C00567 V=800.0 PL=0
MOVL C00568 V=800.0 PL=0
MOVL C00569 V=800.0 PL=0
MOVL C00570 V=800.0 PL=0
MOVL C00571 V=800.0 PL=0
MOVL C00572 V=800.0 PL=0
MOVL C00573 V=800.0 PL=0
MOVL C00574 V=800.0 PL=0
MOVL C00575 V=800.0 PL=0
MOVL C00576 V=800.0 PL=0
MOVL C00577 V=800.0 PL=0
MOVL C00578 V=800.0 PL=0
MOVL C00579 V=800.0 PL=0
MOVL C00580 V=800.0 PL=0
MOVL C00581 V=800.0 PL=0
MOVL C00582 V=800.0 PL=0
MOVL C00583 V=800.0 PL=0
MOVL C00584 V=800.0 PL=0
MOVL C00585 V=800.0 PL=0
MOVL C00586 V=800.0 PL=0
MOVL C00587 V=800.0 PL=0
MOVL C00588 V=800.0 PL=0
MOVL C00589 V=800.0 PL=0
MOVL C00590 V=800.0 PL=0
MOVL C00591 V=800.0 PL=0
MOVL C00592 V=800.0 PL=0
MOVL C00593 V=800.0 PL=0
MOVL C00594 V=800.0 PL=0
MOVL C00595 V=800.0 PL=0
MOVL C00596 V=800.0 PL=0
MOVL C00597 V=800.0 PL=0
MOVL C00598 V=800.0 PL=0
MOVL C00599 V=800.0 PL=0
MOVL C00600 V=800.0 PL=0
MOVL C00601 V=800.0 PL=0
MOVL C00602 V=800.0 PL=0
MOVL C00603 V=800.0 PL=0
MOVL C00604 V=800.0 PL=0
MOVL C00605 V=800.0 PL=0
MOVL C00606 V=800.0 PL=0
MOVL C00607 V=800.0 PL=0
MOVL C00608 V=800.0 PL=0
MOVL C00609 V=800.0 PL=0
MOVL C00610 V=800.0 PL=0
MOVL C00611 V=800.0 PL=0
MOVL C00612 V=800.0 PL=0
MOVL C00613 V=800.0 PL=0
MOVL C00614 V=800.0 PL=0
MOVL C00615 V=800.0 PL=0
MOVL C00616 V=800.0 PL=0
MOVL C00617 V=800.0 PL=0
MOVL C00618 V=800.0 PL=0
MOVL C00619 V=800.0 PL=0
MOVL C00620 V=800.0 PL=0
MOVL C00621 V=800.0 PL=0
MOVL C00622 V=800.0 PL=0
MOVL C00623 V=800.0 PL=0
MOVL C00624 V=800.0 PL=0
MOVL C00625 V=800.0 PL=0
MOVL C00626 V=800.0 PL=0
MOVL C00627 V=800.0 PL=0
MOVL C00628 V=800.0 PL=0
MOVL C00629 V=800.0 PL=0
MOVL C00630 V=800.0 PL=0
MOVL C00631 V=800.0 PL=0
MOVL C00632 V=800.0 PL=0
MOVL C00633 V=800.0 PL=0
MOVL C00634 V=800.0 PL=0
MOVL C00635 V=800.0 PL=0
MOVL C00636 V=800.0 PL=0
MOVL C00637 V=800.0 PL=0
MOVL C00638 V=800.0 PL=0
MOVL C00639 V=800.0 PL=0
MOVL C00640 V=800.0 PL=0
MOVL C00641 V=800.0 PL=0
MOVL C00642 V=800.0 PL=0
MOVL C00643 V=800.0 PL=0
MOVL C00644 V=800.0 PL=0
MOVL C00645 V=800.0 PL=0
MOVL C00646 V=800.0 PL=0
MOVL C00647 V=800.0 PL=0
MOVL C00648 V=800.0 PL=0
MOVL C00649 V=800.0 PL=0
MOVL C00650 V=800.0 PL=0
MOVL C00651 V=800.0 PL=0
MOVL C00652 V=800.0 PL=0
MOVL C00653 V=800.0 PL=0
MOVL C00654 V=800.0 PL=0
MOVL C00655 V=800.0 PL=0
MOVL C00656 V=800.0 PL=0
MOVL C00657 V=800.0 PL=0
MOVL C00658 V=800.0 PL=0
MOVL C00659 V=800.0 PL=0
MOVL C00660 V=800.0 PL=0
MOVL C00661 V=800.0 PL=0
MOVL C00662 V=800.0 PL=0
MOVL C00663 V=800.0 PL=0
MOVL C00664 V=800.0 PL=0
MOVL C00665 V=800.0 PL=0
MOVL C00666 V=800.0 PL=0
MOVL C00667 V=800.0 PL=0
MOVL C00668 V=800.0 PL=0
MOVL C00669 V=800.0 PL=0
MOVL C00670 V=800.0 PL=0
MOVL C00671 V=800.0 PL=0
MOVL C00672 V=800.0 PL=0
MOVL C00673 V=800.0 PL=0
MOVL C00674 V=800.0 PL=0
MOVL C00675 V=800.0 PL=0
MOVL C00676 V=800.0 PL=0
MOVL C00677 V=800.0 PL=0
MOVL C00678 V=800.0 PL=0
MOVL C00679 V=800.0 PL=0
MOVL C00680 V=800.0 PL=0
MOVL C00681 V=800.0 PL=0
MOVL C00682 V=800.0 PL=0
MOVL C00683 V=800.0 PL=0
MOVL C00684 V=800.0 PL=0
MOVL C00685 V=800.0 PL=0
MOVL C00686 V=800.0 PL=0
MOVL C00687 V=800.0 PL=0
MOVL C00688 V=800.0 PL=0
MOVL C00689 V=800.0 PL=0
MOVL C00690 V=800.0 PL=0
MOVL C00691 V=800.0 PL=0
MOVL C00692 V=800.0 PL=0
MOVL C00693 V=800.0 PL=0
MOVL C00694 V=800.0 PL=0
MOVL C00695 V=800.0 PL=0
MOVL C00696 V=800.0 PL=0
MOVL C00697 V=800.0 PL=0
MOVL C00698 V=800.0 PL=0
MOVL C00699 V=800.0 PL=0
MOVL C00700 V=800.0 PL=0
MOVL C00701 V=800.0 PL=0
MOVL C00702 V=800.0 PL=0
MOVL C00703 V=800.0 PL=0
MOVL C00704 V=800.0 PL=0
MOVL C00705 V=800.0 PL=0
MOVL C00706 V=800.0 PL=0
MOVL C00707 V=800.0 PL=0
MOVL C00708 V=800.0 PL=0
MOVL C00709 V=800.0 PL=0
MOVL C00710 V=800.0 PL=0
MOVL C00711 V=800.0 PL=0
MOVL C00712 V=800.0 PL=0
MOVL C00713 V=800.0 PL=0
MOVL C00714 V=800.0 PL=0
MOVL C00715 V=800.0 PL=0
MOVL C00716 V=800.0 PL=0
MOVL C00717 V=800.0 PL=0
MOVL C00718 V=800.0 PL=0
MOVL C00719 V=800.0 PL=0
MOVL C00720 V=800.0 PL=0
MOVL C00721 V=800.0 PL=0
MOVL C00722 V=800.0 PL=0
MOVL C00723 V=800.0 PL=0
MOVL C00724 V=800.0 PL=0
MOVL C00725 V=800.0 PL=0
MOVL C00726 V=800.0 PL=0
MOVL C00727 V=800.0 PL=0
MOVL C00728 V=800.0 PL=0
MOVL C00729 V=800.0 PL=0
MOVL C00730 V=800.0 PL=0
MOVL C00731 V=800.0 PL=0
MOVL C00732 V=800.0 PL=0
MOVL C00733 V=800.0 PL=0
MOVL C00734 V=800.0 PL=0
MOVL C00735 V=800.0 PL=0
MOVL C00736 V=800.0 PL=0
MOVL C00737 V=800.0 PL=0
MOVL C00738 V=800.0 PL=0
MOVL C00739 V=800.0 PL=0
MOVL C00740 V=800.0 PL=0
MOVL C00741 V=800.0 PL=0
MOVL C00742 V=800.0 PL=0
MOVL C00743 V=800.0 PL=0
MOVL C00744 V=800.0 PL=0
MOVL C00745 V=800.0 PL=0
MOVL C00746 V=800.0 PL=0
MOVL C00747 V=800.0 PL=0
MOVL C00748 V=800.0 PL=0
MOVL C00749 V=800.0 PL=0
MOVL C00750 V=800.0 PL=0
MOVL C00751 V=800.0 PL=0
MOVL C00752 V=800.0 PL=0
MOVL C00753 V=800.0 PL=0
MOVL C00754 V=800.0 PL=0
MOVL C00755 V=800.0 PL=0
MOVL C00756 V=800.0 PL=0
MOVL C00757 V=800.0 PL=0
MOVL C00758 V=800.0 PL=0
MOVL C00759 V=800.0 PL=0
MOVL C00760 V=800.0 PL=0
MOVL C00761 V=800.0 PL=0
MOVL C00762 V=800.0 PL=0
MOVL C00763 V=800.0 PL=0
MOVL C00764 V=800.0 PL=0
MOVL C00765 V=800.0 PL=0
MOVL C00766 V=800.0 PL=0
MOVL C00767 V=800.0 PL=0
MOVL C00768 V=800.0 PL=0
MOVL C00769 V=800.0 PL=0
MOVL C00770 V=800.0 PL=0
MOVL C00771 V=800.0 PL=0
MOVL C00772 V=800.0 PL=0
MOVL C00773 V=800.0 PL=0
MOVL C00774 V=800.0 PL=0
MOVL C00775 V=800.0 PL=0
MOVL C00776 V=800.0 PL=0
MOVL C00777 V=800.0 PL=0
MOVL C00778 V=800.0 PL=0
MOVL C00779 V=800.0 PL=0
MOVL C00780 V=800.0 PL=0
MOVL C00781 V=800.0 PL=0
MOVL C00782 V=800.0 PL=0
MOVL C00783 V=800.0 PL=0
MOVL C00784 V=800.0 PL=0
MOVL C00785 V=800.0 PL=0
MOVL C00786 V=800.0 PL=0
MOVL C00787 V=800.0 PL=0
MOVL C00788 V=800.0 PL=0
MOVL C00789 V=800.0 PL=0
MOVL C00790 V=800.0 PL=0
MOVL C00791 V=800.0 PL=0
MOVL C00792 V=800.0 PL=0
MOVL C00793 V=800.0 PL=0
MOVL C00794 V=800.0 PL=0
MOVL C00795 V=800.0 PL=0
MOVL C00796 V=800.0 PL=0
MOVL C00797 V=800.0 PL=0
MOVL C00798 V=800.0 PL=0
MOVL C00799 V=800.0 PL=0
MOVL C00800 V=800.0 PL=0
MOVL C00801 V=800.0 PL=0
MOVL C00802 V=800.0 PL=0
MOVL C00803 V=800.0 PL=0
MOVL C00804 V=800.0 PL=0
MOVL C00805 V=800.0 PL=0
MOVL C00806 V=800.0 PL=0
MOVL C00807 V=800.0 PL=0
MOVL C00808 V=800.0 PL=0
MOVL C00809 V=800.0 PL=0
MOVL C00810 V=800.0 PL=0
MOVL C00811 V=800.0 PL=0
MOVL C00812 V=800.0 PL=0
MOVL C00813 V=800.0 PL=0
MOVL C00814 V=800.0 PL=0
MOVL C00815 V=800.0 PL=0
MOVL C00816 V=800.0 PL=0
MOVL C00817 V=800.0 PL=0
MOVL C00818 V=800.0 PL=0
MOVL C00819 V=800.0 PL=0
MOVL C00820 V=800.0 PL=0
MOVL C00821 V=800.0 PL=0
MOVL C00822 V=800.0 PL=0
MOVL C00823 V=800.0 PL=0
MOVL C00824 V=800.0 PL=0
MOVL C00825 V=800.0 PL=0
MOVL C00826 V=800.0 PL=0
MOVL C00827 V=800.0 PL=0
MOVL C00828 V=800.0 PL=0
MOVL C00829 V=800.0 PL=0
MOVL C00830 V=800.0 PL=0
MOVL C00831 V=800.0 PL=0
MOVL C00832 V=800.0 PL=0
MOVL C00833 V=800.0 PL=0
MOVL C00834 V=800.0 PL=0
MOVL C00835 V=800.0 PL=0
MOVL C00836 V=800.0 PL=0
MOVL C00837 V=800.0 PL=0
MOVL C00838 V=800.0 PL=0
MOVL C00839 V=800.0 PL=0
MOVL C00840 V=800.0 PL=0
MOVL C00841 V=800.0 PL=0
MOVL C00842 V=800.0 PL=0
MOVL C00843 V=800.0 PL=0
MOVL C00844 V=800.0 PL=0
MOVL C00845 V=800.0 PL=0
MOVL C00846 V=800.0 PL=0
MOVL C00847 V=800.0 PL=0
MOVL C00848 V=800.0 PL=0
MOVL C00849 V=800.0 PL=0
MOVL C00850 V=800.0 PL=0
MOVL C00851 V=800.0 PL=0
MOVL C00852 V=800.0 PL=0
MOVL C00853 V=800.0 PL=0
MOVL C00854 V=800.0 PL=0
MOVL C00855 V=800.0 PL=0
MOVL C00856 V=800.0 PL=0
MOVL C00857 V=800.0 PL=0
MOVL C00858 V=800.0 PL=0
MOVL C00859 V=800.0 PL=0
MOVL C00860 V=800.0 PL=0
MOVL C00861 V=800.0 PL=0
MOVL C00862 V=800.0 PL=0
MOVL C00863 V=800.0 PL=0
MOVL C00864 V=800.0 PL=0
MOVL C00865 V=800.0 PL=0
MOVL C00866 V=800.0 PL=0
MOVL C00867 V=800.0 PL=0
MOVL C00868 V=800.0 PL=0
MOVL C00869 V=800.0 PL=0
MOVL C00870 V=800.0 PL=0
MOVL C00871 V=800.0 PL=0
MOVL C00872 V=800.0 PL=0
MOVL C00873 V=800.0 PL=0
MOVL C00874 V=800.0 PL=0
MOVL C00875 V=800.0 PL=0
MOVL C00876 V=800.0 PL=0
MOVL C00877 V=800.0 PL=0
MOVL C00878 V=800.0 PL=0
MOVL C00879 V=800.0 PL=0
MOVL C00880 V=800.0 PL=0
MOVL C00881 V=800.0 PL=0
MOVL C00882 V=800.0 PL=0
MOVL C00883 V=800.0 PL=0
MOVL C00884 V=800.0 PL=0
MOVL C00885 V=800.0 PL=0
MOVL C00886 V=800.0 PL=0
MOVL C00887 V=800.0 PL=0
MOVL C00888 V=800.0 PL=0
MOVL C00889 V=800.0 PL=0
MOVL C00890 V=800.0 PL=0
MOVL C00891 V=800.0 PL=0
MOVL C00892 V=800.0 PL=0
MOVL C00893 V=800.0 PL=0
MOVL C00894 V=800.0 PL=0
MOVL C00895 V=800.0 PL=0
MOVL C00896 V=800.0 PL=0
MOVL C00897 V=800.0 PL=0
MOVL C00898 V=800.0 PL=0
MOVL C00899 V=800.0 PL=0
MOVL C00900 V=800.0 PL=0
MOVL C00901 V=800.0 PL=0
MOVL C00902 V=800.0 PL=0
MOVL C00903 V=800.0 PL=0
MOVL C00904 V=800.0 PL=0
MOVL C00905 V=800.0 PL=0
MOVL C00906 V=800.0 PL=0
MOVL C00907 V=800.0 PL=0
MOVL C00908 V=800.0 PL=0
MOVL C00909 V=800.0 PL=0
MOVL C00910 V=800.0 PL=0
MOVL C00911 V=800.0 PL=0
MOVL C00912 V=800.0 PL=0
MOVL C00913 V=800.0 PL=0
MOVL C00914 V=800.0 PL=0
MOVL C00915 V=800.0 PL=0
MOVL C00916 V=800.0 PL=0
MOVL C00917 V=800.0 PL=0
MOVL C00918 V=800.0 PL=0
MOVL C00919 V=800.0 PL=0
MOVL C00920 V=800.0 PL=0
MOVL C00921 V=800.0 PL=0
MOVL C00922 V=800.0 PL=0
MOVL C00923 V=800.0 PL=0
MOVL C00924 V=800.0 PL=0
MOVL C00925 V=800.0 PL=0
MOVL C00926 V=800.0 PL=0
MOVL C00927 V=800.0 PL=0
MOVL C00928 V=800.0 PL=0
MOVL C00929 V=800.0 PL=0
MOVL C00930 V=800.0 PL=0
MOVL C00931 V=800.0 PL=0
MOVL C00932 V=800.0 PL=0
MOVL C00933 V=800.0 PL=0
MOVL C00934 V=800.0 PL=0
MOVL C00935 V=800.0 PL=0
MOVL C00936 V=800.0 PL=0
MOVL C00937 V=800.0 PL=0
MOVL C00938 V=800.0 PL=0
MOVL C00939 V=800.0 PL=0
MOVL C00940 V=800.0 PL=0
MOVL C00941 V=800.0 PL=0
MOVL C00942 V=800.0 PL=0
MOVL C00943 V=800.0 PL=0
MOVL C00944 V=800.0 PL=0
MOVL C00945 V=800.0 PL=0
MOVL C00946 V=800.0 PL=0
MOVL C00947 V=800.0 PL=0
MOVL C00948 V=800.0 PL=0
MOVL C00949 V=800.0 PL=0
MOVL C00950 V=800.0 PL=0
MOVL C00951 V=800.0 PL=0
MOVL C00952 V=800.0 PL=0
MOVL C00953 V=800.0 PL=0
MOVL C00954 V=800.0 PL=0
MOVL C00955 V=800.0 PL=0
MOVL C00956 V=800.0 PL=0
MOVL C00957 V=800.0 PL=0
MOVL C00958 V=800.0 PL=0
MOVL C00959 V=800.0 PL=0
MOVL C00960 V=800.0 PL=0
MOVL C00961 V=800.0 PL=0
MOVL C00962 V=800.0 PL=0
MOVL C00963 V=800.0 PL=0
MOVL C00964 V=800.0 PL=0
MOVL C00965 V=800.0 PL=0
MOVL C00966 V=800.0 PL=0
MOVL C00967 V=800.0 PL=0
MOVL C00968 V=800.0 PL=0
MOVL C00969 V=800.0 PL=0
MOVL C00970 V=800.0 PL=0
MOVL C00971 V=800.0 PL=0
MOVL C00972 V=800.0 PL=0
MOVL C00973 V=800.0 PL=0
MOVL C00974 V=800.0 PL=0
MOVL C00975 V=800.0 PL=0
MOVL C00976 V=800.0 PL=0
MOVL C00977 V=800.0 PL=0
MOVL C00978 V=800.0 PL=0
MOVL C00979 V=800.0 PL=0
MOVL C00980 V=800.0 PL=0
MOVL C00981 V=800.0 PL=0
MOVL C00982 V=800.0 PL=0
MOVL C00983 V=800.0 PL=0
MOVL C00984 V=800.0 PL=0
MOVL C00985 V=800.0 PL=0
MOVL C00986 V=800.0 PL=0
MOVL C00987 V=800.0 PL=0
MOVL C00988 V=800.0 PL=0
MOVL C00989 V=800.0 PL=0
MOVL C00990 V=800.0 PL=0
MOVL C00991 V=800.0 PL=0
MOVL C00992 V=800.0 PL=0
MOVL C00993 V=800.0 PL=0
MOVL C00994 V=800.0 PL=0
MOVL C00995 V=800.0 PL=0
MOVL C00996 V=800.0 PL=0
MOVL C00997 V=800.0 PL=0
MOVL C00998 V=800.0 PL=0
MOVL C00999 V=800.0 PL=0
MOVL C01000 V=800.0 PL=0
MOVL C01001 V=800.0 PL=0
MOVL C01002 V=800.0 PL=0
MOVL C01003 V=800.0 PL=0
MOVL C01004 V=800.0 PL=0
MOVL C01005 V=800.0 PL=0
MOVL C01006 V=800.0 PL=0
MOVL C01007 V=800.0 PL=0
MOVL C01008 V=800.0 PL=0
MOVL C01009 V=800.0 PL=0
MOVL C01010 V=800.0 PL=0
MOVL C01011 V=800.0 PL=0
MOVL C01012 V=800.0 PL=0
MOVL C01013 V=800.0 PL=0
MOVL C01014 V=800.0 PL=0
MOVL C01015 V=800.0 PL=0
MOVL C01016 V=800.0 PL=0
MOVL C01017 V=800.0 PL=0
MOVL C01018 V=800.0 PL=0
MOVL C01019 V=800.0 PL=0
MOVL C01020 V=800.0 PL=0
MOVL C01021 V=800.0 PL=0
MOVL C01022 V=800.0 PL=0
MOVL C01023 V=800.0 PL=0
MOVL C01024 V=800.0 PL=0
MOVL C01025 V=800.0 PL=0
MOVL C01026 V=800.0 PL=0
MOVL C01027 V=800.0 PL=0
MOVL C01028 V=800.0 PL=0
MOVL C01029 V=800.0 PL=0
MOVL C01030 V=800.0 PL=0
MOVL C01031 V=800.0 PL=0
MOVL C01032 V=800.0 PL=0
MOVL C01033 V=800.0 PL=0
MOVL C01034 V=800.0 PL=0
MOVL C01035 V=800.0 PL=0
MOVL C01036 V=800.0 PL=0
MOVL C01037 V=800.0 PL=0
MOVL C01038 V=800.0 PL=0
MOVL C01039 V=800.0 PL=0
MOVL C01040 V=800.0 PL=0
MOVL C01041 V=800.0 PL=0
MOVL C01042 V=800.0 PL=0
MOVL C01043 V=800.0 PL=0
MOVL C01044 V=800.0 PL=0
MOVL C01045 V=800.0 PL=0
MOVL C01046 V=800.0 PL=0
MOVL C01047 V=800.0 PL=0
MOVL C01048 V=800.0 PL=0
MOVL C01049 V=800.0 PL=0
MOVL C01050 V=800.0 PL=0
MOVL C01051 V=800.0 PL=0
MOVL C01052 V=800.0 PL=0
MOVL C01053 V=800.0 PL=0
MOVL C01054 V=800.0 PL=0
MOVL C01055 V=800.0 PL=0
MOVL C01056 V=800.0 PL=0
MOVL C01057 V=800.0 PL=0
MOVL C01058 V=800.0 PL=0
MOVL C01059 V=800.0 PL=0
MOVL C01060 V=800.0 PL=0
MOVL C01061 V=800.0 PL=0
MOVL C01062 V=800.0 PL=0
MOVL C01063 V=800.0 PL=0
MOVL C01064 V=800.0 PL=0
MOVL C01065 V=800.0 PL=0
MOVL C01066 V=800.0 PL=0
MOVL C01067 V=800.0 PL=0
MOVL C01068 V=800.0 PL=0
MOVL C01069 V=800.0 PL=0
MOVL C01070 V=800.0 PL=0
MOVL C01071 V=800.0 PL=0
MOVL C01072 V=800.0 PL=0
MOVL C01073 V=800.0 PL=0
MOVL C01074 V=800.0 PL=0
MOVL C01075 V=800.0 PL=0
MOVL C01076 V=800.0 PL=0
MOVL C01077 V=800.0 PL=0
MOVL C01078 V=800.0 PL=0
MOVL C01079 V=800.0 PL=0
MOVL C01080 V=800.0 PL=0
MOVL C01081 V=800.0 PL=0
MOVL C01082 V=800.0 PL=0
MOVL C01083 V=800.0 PL=0
MOVL C01084 V=800.0 PL=0
MOVL C01085 V=800.0 PL=0
MOVL C01086 V=800.0 PL=0
MOVL C01087 V=800.0 PL=0
MOVL C01088 V=800.0 PL=0
MOVL C01089 V=800.0 PL=0
MOVL C01090 V=800.0 PL=0
MOVL C01091 V=800.0 PL=0
MOVL C01092 V=800.0 PL=0
MOVL C01093 V=800.0 PL=0
MOVL C01094 V=800.0 PL=0
MOVL C01095 V=800.0 PL=0
MOVL C01096 V=800.0 PL=0
MOVL C01097 V=800.0 PL=0
MOVL C01098 V=800.0 PL=0
MOVL C01099 V=800.0 PL=0
MOVL C01100 V=800.0 PL=0
MOVL C01101 V=800.0 PL=0
MOVL C01102 V=800.0 PL=0
MOVL C01103 V=800.0 PL=0
MOVL C01104 V=800.0 PL=0
MOVL C01105 V=800.0 PL=0
MOVL C01106 V=800.0 PL=0
MOVL C01107 V=800.0 PL=0
MOVL C01108 V=800.0 PL=0
MOVL C01109 V=800.0 PL=0
MOVL C01110 V=800.0 PL=0
MOVL C01111 V=800.0 PL=0
MOVL C01112 V=800.0 PL=0
MOVL C01113 V=800.0 PL=0
MOVL C01114 V=800.0 PL=0
MOVL C01115 V=800.0 PL=0
MOVL C01116 V=800.0 PL=0
MOVL C01117 V=800.0 PL=0
MOVL C01118 V=800.0 PL=0
MOVL C01119 V=800.0 PL=0
MOVL C01120 V=800.0 PL=0
MOVL C01121 V=800.0 PL=0
MOVL C01122 V=800.0 PL=0
MOVL C01123 V=800.0 PL=0
MOVL C01124 V=800.0 PL=0
MOVL C01125 V=800.0 PL=0
MOVL C01126 V=800.0 PL=0
MOVL C01127 V=800.0 PL=0
MOVL C01128 V=800.0 PL=0
MOVL C01129 V=800.0 PL=0
MOVL C01130 V=800.0 PL=0
MOVL C01131 V=800.0 PL=0
MOVL C01132 V=800.0 PL=0
MOVL C01133 V=800.0 PL=0
MOVL C01134 V=800.0 PL=0
MOVL C01135 V=800.0 PL=0
MOVL C01136 V=800.0 PL=0
MOVL C01137 V=800.0 PL=0
MOVL C01138 V=800.0 PL=0
MOVL C01139 V=800.0 PL=0
MOVL C01140 V=800.0 PL=0
MOVL C01141 V=800.0 PL=0
MOVL C01142 V=800.0 PL=0
MOVL C01143 V=800.0 PL=0
MOVL C01144 V=800.0 PL=0
MOVL C01145 V=800.0 PL=0
MOVL C01146 V=800.0 PL=0
MOVL C01147 V=800.0 PL=0
MOVL C01148 V=800.0 PL=0
MOVL C01149 V=800.0 PL=0
MOVL C01150 V=800.0 PL=0
MOVL C01151 V=800.0 PL=0
MOVL C01152 V=800.0 PL=0
MOVL C01153 V=800.0 PL=0
MOVL C01154 V=800.0 PL=0
MOVL C01155 V=800.0 PL=0
MOVL C01156 V=800.0 PL=0
MOVL C01157 V=800.0 PL=0
MOVL C01158 V=800.0 PL=0
MOVL C01159 V=800.0 PL=0
MOVL C01160 V=800.0 PL=0
MOVL C01161 V=800.0 PL=0
MOVL C01162 V=800.0 PL=0
MOVL C01163 V=800.0 PL=0
MOVL C01164 V=800.0 PL=0
MOVL C01165 V=800.0 PL=0
MOVL C01166 V=800.0 PL=0
MOVL C01167 V=800.0 PL=0
MOVL C01168 V=800.0 PL=0
MOVL C01169 V=800.0 PL=0
MOVL C01170 V=800.0 PL=0
MOVL C01171 V=800.0 PL=0
MOVL C01172 V=800.0 PL=0
MOVL C01173 V=800.0 PL=0
MOVL C01174 V=800.0 PL=0
MOVL C01175 V=800.0 PL=0
MOVL C01176 V=800.0 PL=0
MOVL C01177 V=800.0 PL=0
MOVL C01178 V=800.0 PL=0
MOVL C01179 V=800.0 PL=0
MOVL C01180 V=800.0 PL=0
MOVL C01181 V=800.0 PL=0
MOVL C01182 V=800.0 PL=0
MOVL C01183 V=800.0 PL=0
MOVL C01184 V=800.0 PL=0
MOVL C01185 V=800.0 PL=0
MOVL C01186 V=800.0 PL=0
MOVL C01187 V=800.0 PL=0
MOVL C01188 V=800.0 PL=0
MOVL C01189 V=800.0 PL=0
MOVL C01190 V=800.0 PL=0
MOVL C01191 V=800.0 PL=0
MOVL C01192 V=800.0 PL=0
MOVL C01193 V=800.0 PL=0
MOVL C01194 V=800.0 PL=0
MOVL C01195 V=800.0 PL=0
MOVL C01196 V=800.0 PL=0
MOVL C01197 V=800.0 PL=0
MOVL C01198 V=800.0 PL=0
MOVL C01199 V=800.0 PL=0
MOVL C01200 V=800.0 PL=0
MOVL C01201 V=800.0 PL=0
MOVL C01202 V=800.0 PL=0
MOVL C01203 V=800.0 PL=0
MOVL C01204 V=800.0 PL=0
MOVL C01205 V=800.0 PL=0
MOVL C01206 V=800.0 PL=0
MOVL C01207 V=800.0 PL=0
MOVL C01208 V=800.0 PL=0
MOVL C01209 V=800.0 PL=0
MOVL C01210 V=800.0 PL=0
MOVL C01211 V=800.0 PL=0
MOVL C01212 V=800.0 PL=0
MOVL C01213 V=800.0 PL=0
MOVL C01214 V=800.0 PL=0
MOVL C01215 V=800.0 PL=0
MOVL C01216 V=800.0 PL=0
MOVL C01217 V=800.0 PL=0
MOVL C01218 V=800.0 PL=0
MOVL C01219 V=800.0 PL=0
MOVL C01220 V=800.0 PL=0
MOVL C01221 V=800.0 PL=0
MOVL C01222 V=800.0 PL=0
MOVL C01223 V=800.0 PL=0
MOVL C01224 V=800.0 PL=0
MOVL C01225 V=800.0 PL=0
MOVL C01226 V=800.0 PL=0
MOVL C01227 V=800.0 PL=0
MOVL C01228 V=800.0 PL=0
MOVL C01229 V=800.0 PL=0
MOVL C01230 V=800.0 PL=0
MOVL C01231 V=800.0 PL=0
MOVL C01232 V=800.0 PL=0
MOVL C01233 V=800.0 PL=0
MOVL C01234 V=800.0 PL=0
MOVL C01235 V=800.0 PL=0
MOVL C01236 V=800.0 PL=0
MOVL C01237 V=800.0 PL=0
MOVL C01238 V=800.0 PL=0
MOVL C01239 V=800.0 PL=0
MOVL C01240 V=800.0 PL=0
MOVL C01241 V=800.0 PL=0
MOVL C01242 V=800.0 PL=0
MOVL C01243 V=800.0 PL=0
MOVL C01244 V=800.0 PL=0
MOVL C01245 V=800.0 PL=0
MOVL C01246 V=800.0 PL=0
MOVL C01247 V=800.0 PL=0
MOVL C01248 V=800.0 PL=0
MOVL C01249 V=800.0 PL=0
MOVL C01250 V=800.0 PL=0
MOVL C01251 V=800.0 PL=0
MOVL C01252 V=800.0 PL=0
MOVL C01253 V=800.0 PL=0
MOVL C01254 V=800.0 PL=0
MOVL C01255 V=800.0 PL=0
MOVL C01256 V=800.0 PL=0
MOVL C01257 V=800.0 PL=0
MOVL C01258 V=800.0 PL=0
MOVL C01259 V=800.0 PL=0
MOVL C01260 V=800.0 PL=0
MOVL C01261 V=800.0 PL=0
MOVL C01262 V=800.0 PL=0
MOVL C01263 V=800.0 PL=0
MOVL C01264 V=800.0 PL=0
MOVL C01265 V=800.0 PL=0
MOVL C01266 V=800.0 PL=0
MOVL C01267 V=800.0 PL=0
MOVL C01268 V=800.0 PL=0
MOVL C01269 V=800.0 PL=0
MOVL C01270 V=800.0 PL=0
MOVL C01271 V=800.0 PL=0
MOVL C01272 V=800.0 PL=0
MOVL C01273 V=800.0 PL=0
MOVL C01274 V=800.0 PL=0
MOVL C01275 V=800.0 PL=0
MOVL C01276 V=800.0 PL=0
MOVL C01277 V=800.0 PL=0
MOVL C01278 V=800.0 PL=0
MOVL C01279 V=800.0 PL=0
MOVL C01280 V=800.0 PL=0
MOVL C01281 V=800.0 PL=0
MOVL C01282 V=800.0 PL=0
MOVL C01283 V=800.0 PL=0
MOVL C01284 V=800.0 PL=0
MOVL C01285 V=800.0 PL=0
MOVL C01286 V=800.0 PL=0
MOVL C01287 V=800.0 PL=0
MOVL C01288 V=800.0 PL=0
MOVL C01289 V=800.0 PL=0
MOVL C01290 V=800.0 PL=0
MOVL C01291 V=800.0 PL=0
MOVL C01292 V=800.0 PL=0
MOVL C01293 V=800.0 PL=0
MOVL C01294 V=800.0 PL=0
MOVL C01295 V=800.0 PL=0
MOVL C01296 V=800.0 PL=0
MOVL C01297 V=800.0 PL=0
MOVL C01298 V=800.0 PL=0
MOVL C01299 V=800.0 PL=0
MOVL C01300 V=800.0 PL=0
MOVL C01301 V=800.0 PL=0
MOVL C01302 V=800.0 PL=0
MOVL C01303 V=800.0 PL=0
MOVL C01304 V=800.0 PL=0
MOVL C01305 V=800.0 PL=0
MOVL C01306 V=800.0 PL=0
MOVL C01307 V=800.0 PL=0
MOVL C01308 V=800.0 PL=0
MOVL C01309 V=800.0 PL=0
MOVL C01310 V=800.0 PL=0
MOVL C01311 V=800.0 PL=0
MOVL C01312 V=800.0 PL=0
MOVL C01313 V=800.0 PL=0
MOVL C01314 V=800.0 PL=0
MOVL C01315 V=800.0 PL=0
MOVL C01316 V=800.0 PL=0
MOVL C01317 V=800.0 PL=0
MOVL C01318 V=800.0 PL=0
MOVL C01319 V=800.0 PL=0
MOVL C01320 V=800.0 PL=0
MOVL C01321 V=800.0 PL=0
MOVL C01322 V=800.0 PL=0
MOVL C01323 V=800.0 PL=0
MOVL C01324 V=800.0 PL=0
MOVL C01325 V=800.0 PL=0
MOVL C01326 V=800.0 PL=0
MOVL C01327 V=800.0 PL=0
MOVL C01328 V=800.0 PL=0
MOVL C01329 V=800.0 PL=0
MOVL C01330 V=800.0 PL=0
MOVL C01331 V=800.0 PL=0
MOVL C01332 V=800.0 PL=0
MOVL C01333 V=800.0 PL=0
MOVL C01334 V=800.0 PL=0
MOVL C01335 V=800.0 PL=0
MOVL C01336 V=800.0 PL=0
MOVL C01337 V=800.0 PL=0
MOVL C01338 V=800.0 PL=0
MOVL C01339 V=800.0 PL=0
MOVL C01340 V=800.0 PL=0
MOVL C01341 V=800.0 PL=0
MOVL C01342 V=800.0 PL=0
MOVL C01343 V=800.0 PL=0
MOVL C01344 V=800.0 PL=0
MOVL C01345 V=800.0 PL=0
MOVL C01346 V=800.0 PL=0
MOVL C01347 V=800.0 PL=0
MOVL C01348 V=800.0 PL=0
MOVL C01349 V=800.0 PL=0
MOVL C01350 V=800.0 PL=0
MOVL C01351 V=800.0 PL=0
MOVL C01352 V=800.0 PL=0
MOVL C01353 V=800.0 PL=0
MOVL C01354 V=800.0 PL=0
MOVL C01355 V=800.0 PL=0
MOVL C01356 V=800.0 PL=0
MOVL C01357 V=800.0 PL=0
MOVL C01358 V=800.0 PL=0
MOVL C01359 V=800.0 PL=0
MOVL C01360 V=800.0 PL=0
MOVL C01361 V=800.0 PL=0
MOVL C01362 V=800.0 PL=0
MOVL C01363 V=800.0 PL=0
MOVL C01364 V=800.0 PL=0
MOVL C01365 V=800.0 PL=0
MOVL C01366 V=800.0 PL=0
MOVL C01367 V=800.0 PL=0
MOVL C01368 V=800.0 PL=0
MOVL C01369 V=800.0 PL=0
MOVL C01370 V=800.0 PL=0
MOVL C01371 V=800.0 PL=0
MOVL C01372 V=800.0 PL=0
MOVL C01373 V=800.0 PL=0
MOVL C01374 V=800.0 PL=0
MOVL C01375 V=800.0 PL=0
MOVL C01376 V=800.0 PL=0
MOVL C01377 V=800.0 PL=0
MOVL C01378 V=800.0 PL=0
MOVL C01379 V=800.0 PL=0
MOVL C01380 V=800.0 PL=0
MOVL C01381 V=800.0 PL=0
MOVL C01382 V=800.0 PL=0
MOVL C01383 V=800.0 PL=0
MOVL C01384 V=800.0 PL=0
MOVL C01385 V=800.0 PL=0
MOVL C01386 V=800.0 PL=0
MOVL C01387 V=800.0 PL=0
MOVL C01388 V=800.0 PL=0
MOVL C01389 V=800.0 PL=0
MOVL C01390 V=800.0 PL=0
MOVL C01391 V=800.0 PL=0
MOVL C01392 V=800.0 PL=0
MOVL C01393 V=800.0 PL=0
MOVL C01394 V=800.0 PL=0
MOVL C01395 V=800.0 PL=0
MOVL C01396 V=800.0 PL=0
MOVL C01397 V=800.0 PL=0
MOVL C01398 V=800.0 PL=0
MOVL C01399 V=800.0 PL=0
MOVL C01400 V=800.0 PL=0
MOVL C01401 V=800.0 PL=0
MOVL C01402 V=800.0 PL=0
MOVL C01403 V=800.0 PL=0
MOVL C01404 V=800.0 PL=0
MOVL C01405 V=800.0 PL=0
MOVL C01406 V=800.0 PL=0
MOVL C01407 V=800.0 PL=0
MOVL C01408 V=800.0 PL=0
MOVL C01409 V=800.0 PL=0
MOVL C01410 V=800.0 PL=0
MOVL C01411 V=800.0 PL=0
MOVL C01412 V=800.0 PL=0
MOVL C01413 V=800.0 PL=0
MOVL C01414 V=800.0 PL=0
MOVL C01415 V=800.0 PL=0
MOVL C01416 V=800.0 PL=0
MOVL C01417 V=800.0 PL=0
MOVL C01418 V=800.0 PL=0
MOVL C01419 V=800.0 PL=0
MOVL C01420 V=800.0 PL=0
MOVL C01421 V=800.0 PL=0
MOVL C01422 V=800.0 PL=0
MOVL C01423 V=800.0 PL=0
MOVL C01424 V=800.0 PL=0
MOVL C01425 V=800.0 PL=0
MOVL C01426 V=800.0 PL=0
MOVL C01427 V=800.0 PL=0
MOVL C01428 V=800.0 PL=0
MOVL C01429 V=800.0 PL=0
MOVL C01430 V=800.0 PL=0
MOVL C01431 V=800.0 PL=0
MOVL C01432 V=800.0 PL=0
MOVL C01433 V=800.0 PL=0
MOVL C01434 V=800.0 PL=0
MOVL C01435 V=800.0 PL=0
MOVL C01436 V=800.0 PL=0
MOVL C01437 V=800.0 PL=0
MOVL C01438 V=800.0 PL=0
MOVL C01439 V=800.0 PL=0
MOVL C01440 V=800.0 PL=0
MOVL C01441 V=800.0 PL=0
MOVL C01442 V=800.0 PL=0
MOVL C01443 V=800.0 PL=0
MOVL C01444 V=800.0 PL=0
MOVL C01445 V=800.0 PL=0
MOVL C01446 V=800.0 PL=0
MOVL C01447 V=800.0 PL=0
MOVL C01448 V=800.0 PL=0
MOVL C01449 V=800.0 PL=0
MOVL C01450 V=800.0 PL=0
MOVL C01451 V=800.0 PL=0
MOVL C01452 V=800.0 PL=0
MOVL C01453 V=800.0 PL=0
MOVL C01454 V=800.0 PL=0
MOVL C01455 V=800.0 PL=0
MOVL C01456 V=800.0 PL=0
MOVL C01457 V=800.0 PL=0
MOVL C01458 V=800.0 PL=0
MOVL C01459 V=800.0 PL=0
MOVL C01460 V=800.0 PL=0
MOVL C01461 V=800.0 PL=0
MOVL C01462 V=800.0 PL=0
MOVL C01463 V=800.0 PL=0
MOVL C01464 V=800.0 PL=0
MOVL C01465 V=800.0 PL=0
MOVL C01466 V=800.0 PL=0
MOVL C01467 V=800.0 PL=0
MOVL C01468 V=800.0 PL=0
MOVL C01469 V=800.0 PL=0
MOVL C01470 V=800.0 PL=0
MOVL C01471 V=800.0 PL=0
MOVL C01472 V=800.0 PL=0
MOVL C01473 V=800.0 PL=0
MOVL C01474 V=800.0 PL=0
MOVL C01475 V=800.0 PL=0
MOVL C01476 V=800.0 PL=0
MOVL C01477 V=800.0 PL=0
MOVL C01478 V=800.0 PL=0
MOVL C01479 V=800.0 PL=0
MOVL C01480 V=800.0 PL=0
MOVL C01481 V=800.0 PL=0
MOVL C01482 V=800.0 PL=0
MOVL C01483 V=800.0 PL=0
MOVL C01484 V=800.0 PL=0
MOVL C01485 V=800.0 PL=0
MOVL C01486 V=800.0 PL=0
MOVL C01487 V=800.0 PL=0
MOVL C01488 V=800.0 PL=0
MOVL C01489 V=800.0 PL=0
MOVL C01490 V=800.0 PL=0
MOVL C01491 V=800.0 PL=0
MOVL C01492 V=800.0 PL=0
MOVL C01493 V=800.0 PL=0
MOVL C01494 V=800.0 PL=0
MOVL C01495 V=800.0 PL=0
MOVL C01496 V=800.0 PL=0
MOVL C01497 V=800.0 PL=0
MOVL C01498 V=800.0 PL=0
MOVL C01499 V=800.0 PL=0
MOVL C01500 V=800.0 PL=0
MOVL C01501 V=800.0 PL=0
MOVL C01502 V=800.0 PL=0
MOVL C01503 V=800.0 PL=0
MOVL C01504 V=800.0 PL=0
MOVL C01505 V=800.0 PL=0
MOVL C01506 V=800.0 PL=0
MOVL C01507 V=800.0 PL=0
MOVL C01508 V=800.0 PL=0
MOVL C01509 V=800.0 PL=0
MOVL C01510 V=800.0 PL=0
MOVL C01511 V=800.0 PL=0
MOVL C01512 V=800.0 PL=0
MOVL C01513 V=800.0 PL=0
MOVL C01514 V=800.0 PL=0
MOVL C01515 V=800.0 PL=0
MOVL C01516 V=800.0 PL=0
MOVL C01517 V=800.0 PL=0
MOVL C01518 V=800.0 PL=0
MOVL C01519 V=800.0 PL=0
MOVL C01520 V=800.0 PL=0
MOVL C01521 V=800.0 PL=0
MOVL C01522 V=800.0 PL=0
MOVL C01523 V=800.0 PL=0
MOVL C01524 V=800.0 PL=0
MOVL C01525 V=800.0 PL=0
MOVL C01526 V=800.0 PL=0
MOVL C01527 V=800.0 PL=0
MOVL C01528 V=800.0 PL=0
MOVL C01529 V=800.0 PL=0
MOVL C01530 V=800.0 PL=0
MOVL C01531 V=800.0 PL=0
MOVL C01532 V=800.0 PL=0
MOVL C01533 V=800.0 PL=0
MOVL C01534 V=800.0 PL=0
MOVL C01535 V=800.0 PL=0
MOVL C01536 V=800.0 PL=0
MOVL C01537 V=800.0 PL=0
MOVL C01538 V=800.0 PL=0
MOVL C01539 V=800.0 PL=0
MOVL C01540 V=800.0 PL=0
MOVL C01541 V=800.0 PL=0
MOVL C01542 V=800.0 PL=0
MOVL C01543 V=800.0 PL=0
MOVL C01544 V=800.0 PL=0
MOVL C01545 V=800.0 PL=0
MOVL C01546 V=800.0 PL=0
MOVL C01547 V=800.0 PL=0
MOVL C01548 V=800.0 PL=0
MOVL C01549 V=800.0 PL=0
MOVL C01550 V=800.0 PL=0
MOVL C01551 V=800.0 PL=0
MOVL C01552 V=800.0 PL=0
MOVL C01553 V=800.0 PL=0
MOVL C01554 V=800.0 PL=0
MOVL C01555 V=800.0 PL=0
MOVL C01556 V=800.0 PL=0
MOVL C01557 V=800.0 PL=0
MOVL C01558 V=800.0 PL=0
MOVL C01559 V=800.0 PL=0
MOVL C01560 V=800.0 PL=0
MOVL C01561 V=800.0 PL=0
MOVL C01562 V=800.0 PL=0
MOVL C01563 V=800.0 PL=0
MOVL C01564 V=800.0 PL=0
MOVL C01565 V=800.0 PL=0
MOVL C01566 V=800.0 PL=0
MOVL C01567 V=800.0 PL=0
MOVL C01568 V=800.0 PL=0
MOVL C01569 V=800.0 PL=0
MOVL C01570 V=800.0 PL=0
MOVL C01571 V=800.0 PL=0
MOVL C01572 V=800.0 PL=0
MOVL C01573 V=800.0 PL=0
MOVL C01574 V=800.0 PL=0
MOVL C01575 V=800.0 PL=0
MOVL C01576 V=800.0 PL=0
MOVL C01577 V=800.0 PL=0
MOVL C01578 V=800.0 PL=0
MOVL C01579 V=800.0 PL=0
MOVL C01580 V=800.0 PL=0
MOVL C01581 V=800.0 PL=0
MOVL C01582 V=800.0 PL=0
MOVL C01583 V=800.0 PL=0
MOVL C01584 V=800.0 PL=0
MOVL C01585 V=800.0 PL=0
MOVL C01586 V=800.0 PL=0
MOVL C01587 V=800.0 PL=0
MOVL C01588 V=800.0 PL=0
MOVL C01589 V=800.0 PL=0
MOVL C01590 V=800.0 PL=0
MOVL C01591 V=800.0 PL=0
MOVL C01592 V=800.0 PL=0
MOVL C01593 V=800.0 PL=0
MOVL C01594 V=800.0 PL=0
MOVL C01595 V=800.0 PL=0
MOVL C01596 V=800.0 PL=0
MOVL C01597 V=800.0 PL=0
MOVL C01598 V=800.0 PL=0
MOVL C01599 V=800.0 PL=0
MOVL C01600 V=800.0 PL=0
MOVL C01601 V=800.0 PL=0
MOVL C01602 V=800.0 PL=0
MOVL C01603 V=800.0 PL=0
MOVL C01604 V=800.0 PL=0
MOVL C01605 V=800.0 PL=0
MOVL C01606 V=800.0 PL=0
MOVL C01607 V=800.0 PL=0
MOVL C01608 V=800.0 PL=0
MOVL C01609 V=800.0 PL=0
MOVL C01610 V=800.0 PL=0
MOVL C01611 V=800.0 PL=0
MOVL C01612 V=800.0 PL=0
MOVL C01613 V=800.0 PL=0
MOVL C01614 V=800.0 PL=0
MOVL C01615 V=800.0 PL=0
MOVL C01616 V=800.0 PL=0
MOVL C01617 V=800.0 PL=0
MOVL C01618 V=800.0 PL=0
MOVL C01619 V=800.0 PL=0
MOVL C01620 V=800.0 PL=0
MOVL C01621 V=800.0 PL=0
MOVL C01622 V=800.0 PL=0
MOVL C01623 V=800.0 PL=0
MOVL C01624 V=800.0 PL=0
MOVL C01625 V=800.0 PL=0
MOVL C01626 V=800.0 PL=0
MOVL C01627 V=800.0 PL=0
MOVL C01628 V=800.0 PL=0
MOVL C01629 V=800.0 PL=0
MOVL C01630 V=800.0 PL=0
MOVL C01631 V=800.0 PL=0
MOVL C01632 V=800.0 PL=0
MOVL C01633 V=800.0 PL=0
MOVL C01634 V=800.0 PL=0
MOVL C01635 V=800.0 PL=0
MOVL C01636 V=800.0 PL=0
MOVL C01637 V=800.0 PL=0
MOVL C01638 V=800.0 PL=0
MOVL C01639 V=800.0 PL=0
MOVL C01640 V=800.0 PL=0
MOVL C01641 V=800.0 PL=0
MOVL C01642 V=800.0 PL=0
MOVL C01643 V=800.0 PL=0
MOVL C01644 V=800.0 PL=0
MOVL C01645 V=800.0 PL=0
MOVL C01646 V=800.0 PL=0
MOVL C01647 V=800.0 PL=0
MOVL C01648 V=800.0 PL=0
MOVL C01649 V=800.0 PL=0
MOVL C01650 V=800.0 PL=0
MOVL C01651 V=800.0 PL=0
MOVL C01652 V=800.0 PL=0
MOVL C01653 V=800.0 PL=0
MOVL C01654 V=800.0 PL=0
MOVL C01655 V=800.0 PL=0
MOVL C01656 V=800.0 PL=0
MOVL C01657 V=800.0 PL=0
MOVL C01658 V=800.0 PL=0
MOVL C01659 V=800.0 PL=0
MOVL C01660 V=800.0 PL=0
MOVL C01661 V=800.0 PL=0
MOVL C01662 V=800.0 PL=0
MOVL C01663 V=800.0 PL=0
MOVL C01664 V=800.0 PL=0
MOVL C01665 V=800.0 PL=0
MOVL C01666 V=800.0 PL=0
MOVL C01667 V=800.0 PL=0
MOVL C01668 V=800.0 PL=0
MOVL C01669 V=800.0 PL=0
MOVL C01670 V=800.0 PL=0
MOVL C01671 V=800.0 PL=0
MOVL C01672 V=800.0 PL=0
MOVL C01673 V=800.0 PL=0
MOVL C01674 V=800.0 PL=0
MOVL C01675 V=800.0 PL=0
MOVL C01676 V=800.0 PL=0
MOVL C01677 V=800.0 PL=0
MOVL C01678 V=800.0 PL=0
MOVL C01679 V=800.0 PL=0
MOVL C01680 V=800.0 PL=0
MOVL C01681 V=800.0 PL=0
MOVL C01682 V=800.0 PL=0
MOVL C01683 V=800.0 PL=0
MOVL C01684 V=800.0 PL=0
MOVL C01685 V=800.0 PL=0
MOVL C01686 V=800.0 PL=0
MOVL C01687 V=800.0 PL=0
MOVL C01688 V=800.0 PL=0
MOVL C01689 V=800.0 PL=0
MOVL C01690 V=800.0 PL=0
MOVL C01691 V=800.0 PL=0
MOVL C01692 V=800.0 PL=0
MOVL C01693 V=800.0 PL=0
MOVL C01694 V=800.0 PL=0
MOVL C01695 V=800.0 PL=0
MOVL C01696 V=800.0 PL=0
MOVL C01697 V=800.0 PL=0
MOVL C01698 V=800.0 PL=0
MOVL C01699 V=800.0 PL=0
MOVL C01700 V=800.0 PL=0
MOVL C01701 V=800.0 PL=0
MOVL C01702 V=800.0 PL=0
MOVL C01703 V=800.0 PL=0
MOVL C01704 V=800.0 PL=0
MOVL C01705 V=800.0 PL=0
MOVL C01706 V=800.0 PL=0
MOVL C01707 V=800.0 PL=0
MOVL C01708 V=800.0 PL=0
MOVL C01709 V=800.0 PL=0
MOVL C01710 V=800.0 PL=0
MOVL C01711 V=800.0 PL=0
MOVL C01712 V=800.0 PL=0
MOVL C01713 V=800.0 PL=0
MOVL C01714 V=800.0 PL=0
MOVL C01715 V=800.0 PL=0
MOVL C01716 V=800.0 PL=0
MOVL C01717 V=800.0 PL=0
MOVL C01718 V=800.0 PL=0
MOVL C01719 V=800.0 PL=0
MOVL C01720 V=800.0 PL=0
MOVL C01721 V=800.0 PL=0
MOVL C01722 V=800.0 PL=0
MOVL C01723 V=800.0 PL=0
MOVL C01724 V=800.0 PL=0
MOVL C01725 V=800.0 PL=0
MOVL C01726 V=800.0 PL=0
MOVL C01727 V=800.0 PL=0
MOVL C01728 V=800.0 PL=0
MOVL C01729 V=800.0 PL=0
MOVL C01730 V=800.0 PL=0
MOVL C01731 V=800.0 PL=0
MOVL C01732 V=800.0 PL=0
MOVL C01733 V=800.0 PL=0
MOVL C01734 V=800.0 PL=0
MOVL C01735 V=800.0 PL=0
MOVL C01736 V=800.0 PL=0
MOVL C01737 V=800.0 PL=0
MOVL C01738 V=800.0 PL=0
MOVL C01739 V=800.0 PL=0
MOVL C01740 V=800.0 PL=0
MOVL C01741 V=800.0 PL=0
MOVL C01742 V=800.0 PL=0
MOVL C01743 V=800.0 PL=0
MOVL C01744 V=800.0 PL=0
MOVL C01745 V=800.0 PL=0
MOVL C01746 V=800.0 PL=0
MOVL C01747 V=800.0 PL=0
MOVL C01748 V=800.0 PL=0
MOVL C01749 V=800.0 PL=0
MOVL C01750 V=800.0 PL=0
MOVL C01751 V=800.0 PL=0
MOVL C01752 V=800.0 PL=0
MOVL C01753 V=800.0 PL=0
MOVL C01754 V=800.0 PL=0
MOVL C01755 V=800.0 PL=0
MOVL C01756 V=800.0 PL=0
MOVL C01757 V=800.0 PL=0
MOVL C01758 V=800.0 PL=0
MOVL C01759 V=800.0 PL=0
MOVL C01760 V=800.0 PL=0
MOVL C01761 V=800.0 PL=0
MOVL C01762 V=800.0 PL=0
MOVL C01763 V=800.0 PL=0
MOVL C01764 V=800.0 PL=0
MOVL C01765 V=800.0 PL=0
MOVL C01766 V=800.0 PL=0
MOVL C01767 V=800.0 PL=0
MOVL C01768 V=800.0 PL=0
MOVL C01769 V=800.0 PL=0
MOVL C01770 V=800.0 PL=0
MOVL C01771 V=800.0 PL=0
MOVL C01772 V=800.0 PL=0
MOVL C01773 V=800.0 PL=0
MOVL C01774 V=800.0 PL=0
MOVL C01775 V=800.0 PL=0
MOVL C01776 V=800.0 PL=0
MOVL C01777 V=800.0 PL=0
MOVL C01778 V=800.0 PL=0
MOVL C01779 V=800.0 PL=0
MOVL C01780 V=800.0 PL=0
MOVL C01781 V=800.0 PL=0
MOVL C01782 V=800.0 PL=0
MOVL C01783 V=800.0 PL=0
MOVL C01784 V=800.0 PL=0
MOVL C01785 V=800.0 PL=0
MOVL C01786 V=800.0 PL=0
MOVL C01787 V=800.0 PL=0
MOVL C01788 V=800.0 PL=0
MOVL C01789 V=800.0 PL=0
MOVL C01790 V=800.0 PL=0
MOVL C01791 V=800.0 PL=0
MOVL C01792 V=800.0 PL=0
MOVL C01793 V=800.0 PL=0
MOVL C01794 V=800.0 PL=0
MOVL C01795 V=800.0 PL=0
MOVL C01796 V=800.0 PL=0
MOVL C01797 V=800.0 PL=0
MOVL C01798 V=800.0 PL=0
MOVL C01799 V=800.0 PL=0
MOVL C01800 V=800.0 PL=0
MOVL C01801 V=800.0 PL=0
MOVL C01802 V=800.0 PL=0
MOVL C01803 V=800.0 PL=0
MOVL C01804 V=800.0 PL=0
MOVL C01805 V=800.0 PL=0
MOVL C01806 V=800.0 PL=0
MOVL C01807 V=800.0 PL=0
MOVL C01808 V=800.0 PL=0
MOVL C01809 V=800.0 PL=0
MOVL C01810 V=800.0 PL=0
MOVL C01811 V=800.0 PL=0
MOVL C01812 V=800.0 PL=0
MOVL C01813 V=800.0 PL=0
MOVL C01814 V=800.0 PL=0
MOVL C01815 V=800.0 PL=0
MOVL C01816 V=800.0 PL=0
MOVL C01817 V=800.0 PL=0
MOVL C01818 V=800.0 PL=0
MOVL C01819 V=800.0 PL=0
MOVL C01820 V=800.0 PL=0
MOVL C01821 V=800.0 PL=0
MOVL C01822 V=800.0 PL=0
MOVL C01823 V=800.0 PL=0
MOVL C01824 V=800.0 PL=0
MOVL C01825 V=800.0 PL=0
MOVL C01826 V=800.0 PL=0
MOVL C01827 V=800.0 PL=0
MOVL C01828 V=800.0 PL=0
MOVL C01829 V=800.0 PL=0
MOVL C01830 V=800.0 PL=0
MOVL C01831 V=800.0 PL=0
MOVL C01832 V=800.0 PL=0
MOVL C01833 V=800.0 PL=0
MOVL C01834 V=800.0 PL=0
MOVL C01835 V=800.0 PL=0
MOVL C01836 V=800.0 PL=0
MOVL C01837 V=800.0 PL=0
MOVL C01838 V=800.0 PL=0
MOVL C01839 V=800.0 PL=0
MOVL C01840 V=800.0 PL=0
MOVL C01841 V=800.0 PL=0
MOVL C01842 V=800.0 PL=0
MOVL C01843 V=800.0 PL=0
MOVL C01844 V=800.0 PL=0
MOVL C01845 V=800.0 PL=0
MOVL C01846 V=800.0 PL=0
MOVL C01847 V=800.0 PL=0
MOVL C01848 V=800.0 PL=0
MOVL C01849 V=800.0 PL=0
MOVL C01850 V=800.0 PL=0
MOVL C01851 V=800.0 PL=0
MOVL C01852 V=800.0 PL=0
MOVL C01853 V=800.0 PL=0
MOVL C01854 V=800.0 PL=0
MOVL C01855 V=800.0 PL=0
MOVL C01856 V=800.0 PL=0
MOVL C01857 V=800.0 PL=0
MOVL C01858 V=800.0 PL=0
MOVL C01859 V=800.0 PL=0
MOVL C01860 V=800.0 PL=0
MOVL C01861 V=800.0 PL=0
MOVL C01862 V=800.0 PL=0
MOVL C01863 V=800.0 PL=0
MOVL C01864 V=800.0 PL=0
MOVL C01865 V=800.0 PL=0
MOVL C01866 V=800.0 PL=0
MOVL C01867 V=800.0 PL=0
MOVL C01868 V=800.0 PL=0
MOVL C01869 V=800.0 PL=0
MOVL C01870 V=800.0 PL=0
MOVL C01871 V=800.0 PL=0
MOVL C01872 V=800.0 PL=0
MOVL C01873 V=800.0 PL=0
MOVL C01874 V=800.0 PL=0
MOVL C01875 V=800.0 PL=0
MOVL C01876 V=800.0 PL=0
MOVL C01877 V=800.0 PL=0
MOVL C01878 V=800.0 PL=0
MOVL C01879 V=800.0 PL=0
MOVL C01880 V=800.0 PL=0
MOVL C01881 V=800.0 PL=0
MOVL C01882 V=800.0 PL=0
MOVL C01883 V=800.0 PL=0
MOVL C01884 V=800.0 PL=0
MOVL C01885 V=800.0 PL=0
MOVL C01886 V=800.0 PL=0
MOVL C01887 V=800.0 PL=0
MOVL C01888 V=800.0 PL=0
MOVL C01889 V=800.0 PL=0
MOVL C01890 V=800.0 PL=0
MOVL C01891 V=800.0 PL=0
MOVL C01892 V=800.0 PL=0
MOVL C01893 V=800.0 PL=0
MOVL C01894 V=800.0 PL=0
MOVL C01895 V=800.0 PL=0
MOVL C01896 V=800.0 PL=0
MOVL C01897 V=800.0 PL=0
MOVL C01898 V=800.0 PL=0
MOVL C01899 V=800.0 PL=0
MOVL C01900 V=800.0 PL=0
MOVL C01901 V=800.0 PL=0
MOVL C01902 V=800.0 PL=0
MOVL C01903 V=800.0 PL=0
MOVL C01904 V=800.0 PL=0
MOVL C01905 V=800.0 PL=0
MOVL C01906 V=800.0 PL=0
MOVL C01907 V=800.0 PL=0
MOVL C01908 V=800.0 PL=0
MOVL C01909 V=800.0 PL=0
MOVL C01910 V=800.0 PL=0
MOVL C01911 V=800.0 PL=0
MOVL C01912 V=800.0 PL=0
MOVL C01913 V=800.0 PL=0
MOVL C01914 V=800.0 PL=0
MOVL C01915 V=800.0 PL=0
MOVL C01916 V=800.0 PL=0
MOVL C01917 V=800.0 PL=0
MOVL C01918 V=800.0 PL=0
MOVL C01919 V=800.0 PL=0
MOVL C01920 V=800.0 PL=0
MOVL C01921 V=800.0 PL=0
MOVL C01922 V=800.0 PL=0
MOVL C01923 V=800.0 PL=0
MOVL C01924 V=800.0 PL=0
MOVL C01925 V=800.0 PL=0
MOVL C01926 V=800.0 PL=0
MOVL C01927 V=800.0 PL=0
MOVL C01928 V=800.0 PL=0
MOVL C01929 V=800.0 PL=0
MOVL C01930 V=800.0 PL=0
MOVL C01931 V=800.0 PL=0
MOVL C01932 V=800.0 PL=0
MOVL C01933 V=800.0 PL=0
MOVL C01934 V=800.0 PL=0
MOVL C01935 V=800.0 PL=0
MOVL C01936 V=800.0 PL=0
MOVL C01937 V=800.0 PL=0
MOVL C01938 V=800.0 PL=0
MOVL C01939 V=800.0 PL=0
MOVL C01940 V=800.0 PL=0
MOVL C01941 V=800.0 PL=0
MOVL C01942 V=800.0 PL=0
MOVL C01943 V=800.0 PL=0
MOVL C01944 V=800.0 PL=0
MOVL C01945 V=800.0 PL=0
